(* CODESYS project Dashboard.project

Project tree, tasks and I/O mapping:
  Device : CODESYS Control for Raspberry Pi MC SL, CODESYS, order no. 2302000009, version 4.21.0.0
    application Application
      libraries: Standard, 3.5.22.0 (System); ifmEIP, 4.5.1.12 (ifm efector inc.); CAA Memory, * (CAA Technical Workgroup); CAA Can Low Level Extern, * (CAA Technical Workgroup); CmpBitmapPool, * (System)
      task VISU_TASK (cyclic, interval 100 ms, priority 31) calls VisuElems.Visu_Prg
      task MainTask (cyclic, interval t#20ms, priority 1) calls Main
      task ENIPScannerIOTask (cyclic, interval t#10ms, priority 0) calls EtherNet_IP_Scanner.IOCycle
      task ENIPScannerServiceTask (cyclic, interval t#20ms, priority 30) calls EtherNet_IP_Scanner.ServiceCycle
      program Main [ST]
      image pool Logo
      visualisation Connected_Devices_Dashboard
      global variables GL_Variables
      function block IOLink_Dashboard [FBD]: Process_Data, Dashboard_Data
    Onewire
    Ethernet : Ethernet, CODESYS, version 4.2.0.0
        settings: IPAddress = [192,168,1,99]; SubnetMask = [255,255,255,0]; GatewayAddress = [192,168,1,102]; MACAddress = [16#B8,16#27,16#EB,16#2F,16#E3,16#0E]; NetworkInterfaceName = 'eth0'; NetworkInterfaceName = "eth0"; SaveCommunicationSettings = FALSE; IPAddress = [192,168,0,2]; SubnetMask = [255,255,255,0]; GatewayAddress = [0,0,0,0]
      EtherNet_IP_Scanner : EtherNet/IP Scanner, CODESYS, order no. 1, version 4.9.0.0
        AL1423 : IO-Link Master PFL EIP 8P IP69K, ifm electronic, order no. AL1423, version Major Revision=16#2, Minor Revision = 16#3
            settings: INITIALIZED = TRUE; IP address of Target = [16#C0,16#A8,16#01,16#C8]; Keying.Check Minor Revision = FALSE; RequiredConfigVersion = 50660864; Number of Connections = 1; Connection Settings.Requested packet intervall = 10000 µs; Connection Settings.OT Connection Parameters = 18740; Connection Settings.TO Connection Parameters = 18880; Connection Settings.Connection Flags = 1056; Connection Settings.Connection Path Size = 8; Connection Settings.Config#2 Size = 130; Connection Settings.Large OT Connection Parameters = 1207959860; Connection Settings.Large TO Connection Parameters = 1207960000; Heartbeat Multiplier = 1; Input Data.ReadOnly = False; Input Data.BitSize = 16; Input Data.DataSize = 2; Input Data.ReadOnly = False; Input Data.BitSize = 16; Input Data.DataSize = 2; Input Data.ReadOnly = False; Input Data.BitSize = 16; Input Data.DataSize = 2; Input Data.ReadOnly = False; Input Data.BitSize = 16; Input Data.DataSize = 2; Input Data.ReadOnly = False; Input Data.BitSize = 16; Input Data.DataSize = 2; Input Data.ReadOnly = False; Input Data.BitSize = 16; Input Data.DataSize = 2; Input Data.ReadOnly = False; Input Data.BitSize = 16; Input Data.DataSize = 2; Input Data.ReadOnly = False; Input Data.BitSize = 16; Input Data.DataSize = 2; Input Data.ReadOnly = False; Input Data.BitSize = 16;
              Input Data.DataSize = 2; Input Data.ReadOnly = False; Input Data.BitSize = 16; Input Data.DataSize = 2; Input Data.ReadOnly = False; Input Data.BitSize = 16; Input Data.DataSize = 2; Input Data.ReadOnly = False; Input Data.BitSize = 16; Input Data.DataSize = 2; Input Data.ReadOnly = False; Input Data.BitSize = 16; Input Data.DataSize = 2; Input Data.ReadOnly = False; Input Data.BitSize = 16; Input Data.DataSize = 2; Input Data.ReadOnly = False; Input Data.BitSize = 16; Input Data.DataSize = 2; Input Data.ReadOnly = False; Input Data.BitSize = 16; Input Data.DataSize = 2; Input Data.ReadOnly = False; Input Data.BitSize = 16; Input Data.DataSize = 2; Input Data.ReadOnly = False; Input Data.BitSize = 16; Input Data.DataSize = 2; Input Data.ReadOnly = False; Input Data.BitSize = 16; Input Data.DataSize = 2; Input Data.ReadOnly = False; Input Data.BitSize = 16; Input Data.DataSize = 2; Input Data.ReadOnly = False; Input Data.BitSize = 16; Input Data.DataSize = 2; Input Data.ReadOnly = False; Input Data.BitSize = 16; Input Data.DataSize = 2;
              Input Data.ReadOnly = False; Input Data.BitSize = 16; Input Data.DataSize = 2; Input Data.ReadOnly = False; Input Data.BitSize = 16; Input Data.DataSize = 2; Input Data.ReadOnly = False; Input Data.BitSize = 16; Input Data.DataSize = 2; Input Data.ReadOnly = False; Input Data.BitSize = 16; Input Data.DataSize = 2; Input Data.ReadOnly = False; Input Data.BitSize = 16; Input Data.DataSize = 2; Input Data.ReadOnly = False; Input Data.BitSize = 16; Input Data.DataSize = 2; Input Data.ReadOnly = False; Input Data.BitSize = 16; Input Data.DataSize = 2; Input Data.ReadOnly = False; Input Data.BitSize = 16; Input Data.DataSize = 2; Input Data.ReadOnly = False; Input Data.BitSize = 16; Input Data.DataSize = 2; Input Data.ReadOnly = False; Input Data.BitSize = 16; Input Data.DataSize = 2; Input Data.ReadOnly = False; Input Data.BitSize = 16; Input Data.DataSize = 2; Input Data.ReadOnly = False; Input Data.BitSize = 16; Input Data.DataSize = 2; Input Data.ReadOnly = False; Input Data.BitSize = 16; Input Data.DataSize = 2; Input Data.ReadOnly = False;
              Input Data.BitSize = 16; Input Data.DataSize = 2; Input Data.ReadOnly = False; Input Data.BitSize = 16; Input Data.DataSize = 2; Input Data.ReadOnly = False; Input Data.BitSize = 16; Input Data.DataSize = 2; Input Data.ReadOnly = False; Input Data.BitSize = 16; Input Data.DataSize = 2; Input Data.ReadOnly = False; Input Data.BitSize = 16; Input Data.DataSize = 2; Input Data.ReadOnly = False; Input Data.BitSize = 16; Input Data.DataSize = 2; Input Data.ReadOnly = False; Input Data.BitSize = 16; Input Data.DataSize = 2; Input Data.ReadOnly = False; Input Data.BitSize = 16; Input Data.DataSize = 2; Input Data.ReadOnly = False; Input Data.BitSize = 16; Input Data.DataSize = 2; Input Data.ReadOnly = False; Input Data.BitSize = 16; Input Data.DataSize = 2; Input Data.ReadOnly = False; Input Data.BitSize = 16; Input Data.DataSize = 2; Input Data.ReadOnly = False; Input Data.BitSize = 16; Input Data.DataSize = 2; Input Data.ReadOnly = False; Input Data.BitSize = 16; Input Data.DataSize = 2; Input Data.ReadOnly = False; Input Data.BitSize = 16;
              Input Data.DataSize = 2; Input Data.ReadOnly = False; Input Data.BitSize = 16; Input Data.DataSize = 2; Input Data.ReadOnly = False; Input Data.BitSize = 16; Input Data.DataSize = 2; Input Data.ReadOnly = False; Input Data.BitSize = 16; Input Data.DataSize = 2; Input Data.ReadOnly = False; Input Data.BitSize = 16; Input Data.DataSize = 2; Input Data.ReadOnly = False; Input Data.BitSize = 16; Input Data.DataSize = 2; Input Data.ReadOnly = False; Input Data.BitSize = 16; Input Data.DataSize = 2; Input Data.ReadOnly = False; Input Data.BitSize = 16; Input Data.DataSize = 2; Input Data.ReadOnly = False; Input Data.BitSize = 16; Input Data.DataSize = 2; Input Data.ReadOnly = False; Input Data.BitSize = 16; Input Data.DataSize = 2; Input Data.ReadOnly = False; Input Data.BitSize = 16; Input Data.DataSize = 2; Input Data.ReadOnly = False; Input Data.BitSize = 16; Input Data.DataSize = 2; Input Data.ReadOnly = False; Input Data.BitSize = 16; Input Data.DataSize = 2; Input Data.ReadOnly = False; Input Data.BitSize = 16; Input Data.DataSize = 2;
              Input Data.ReadOnly = False; Input Data.BitSize = 16; Input Data.DataSize = 2; Input Data.ReadOnly = False; Input Data.BitSize = 16; Input Data.DataSize = 2; Input Data.ReadOnly = False; Input Data.BitSize = 16; Input Data.DataSize = 2; Input Data.ReadOnly = False; Input Data.BitSize = 16; Input Data.DataSize = 2; Input Data.ReadOnly = False; Input Data.BitSize = 16; Input Data.DataSize = 2; Input Data.ReadOnly = False; Input Data.BitSize = 16; Input Data.DataSize = 2; Input Data.ReadOnly = False; Input Data.BitSize = 16; Input Data.DataSize = 2; Input Data.ReadOnly = False; Input Data.BitSize = 16; Input Data.DataSize = 2; Input Data.ReadOnly = False; Input Data.BitSize = 16; Input Data.DataSize = 2; Input Data.ReadOnly = False; Input Data.BitSize = 16; Input Data.DataSize = 2; Input Data.ReadOnly = False; Input Data.BitSize = 16; Input Data.DataSize = 2; Input Data.ReadOnly = False; Input Data.BitSize = 16; Input Data.DataSize = 2; Input Data.ReadOnly = False; Input Data.BitSize = 16; Input Data.DataSize = 2; Input Data.ReadOnly = False;
              Input Data.BitSize = 16; Input Data.DataSize = 2; Input Data.ReadOnly = False; Input Data.BitSize = 16; Input Data.DataSize = 2; Input Data.ReadOnly = False; Input Data.BitSize = 16; Input Data.DataSize = 2; Input Data.ReadOnly = False; Input Data.BitSize = 16; Input Data.DataSize = 2; Input Data.ReadOnly = False; Input Data.BitSize = 16; Input Data.DataSize = 2; Input Data.ReadOnly = False; Input Data.BitSize = 16; Input Data.DataSize = 2; Input Data.ReadOnly = False; Input Data.BitSize = 16; Input Data.DataSize = 2; Input Data.ReadOnly = False; Input Data.BitSize = 16; Input Data.DataSize = 2; Input Data.ReadOnly = False; Input Data.BitSize = 16; Input Data.DataSize = 2; Input Data.ReadOnly = False; Input Data.BitSize = 16; Input Data.DataSize = 2; Input Data.ReadOnly = False; Input Data.BitSize = 16; Input Data.DataSize = 2; Input Data.ReadOnly = False; Input Data.BitSize = 16; Input Data.DataSize = 2; Input Data.ReadOnly = False; Input Data.BitSize = 16; Input Data.DataSize = 2; Input Data.ReadOnly = False; Input Data.BitSize = 16;
              Input Data.DataSize = 2; Input Data.ReadOnly = False; Input Data.BitSize = 16; Input Data.DataSize = 2; Input Data.ReadOnly = False; Input Data.BitSize = 16; Input Data.DataSize = 2; Input Data.ReadOnly = False; Input Data.BitSize = 16; Input Data.DataSize = 2; Input Data.ReadOnly = False; Input Data.BitSize = 16; Input Data.DataSize = 2; Input Data.ReadOnly = False; Input Data.BitSize = 16; Input Data.DataSize = 2; Input Data.ReadOnly = False; Input Data.BitSize = 16; Input Data.DataSize = 2; Input Data.ReadOnly = False; Input Data.BitSize = 16; Input Data.DataSize = 2; Input Data.ReadOnly = False; Input Data.BitSize = 16; Input Data.DataSize = 2; Input Data.ReadOnly = False; Input Data.BitSize = 16; Input Data.DataSize = 2; Input Data.ReadOnly = False; Input Data.BitSize = 16; Input Data.DataSize = 2; Input Data.ReadOnly = False; Input Data.BitSize = 16; Input Data.DataSize = 2; Input Data.ReadOnly = False; Input Data.BitSize = 16; Input Data.DataSize = 2; Input Data.ReadOnly = False; Input Data.BitSize = 16; Input Data.DataSize = 2;
              Input Data.ReadOnly = False; Input Data.BitSize = 16; Input Data.DataSize = 2; Input Data.ReadOnly = False; Input Data.BitSize = 16; Input Data.DataSize = 2; Input Data.ReadOnly = False; Input Data.BitSize = 16; Input Data.DataSize = 2; Input Data.ReadOnly = False; Input Data.BitSize = 16; Input Data.DataSize = 2; Input Data.ReadOnly = False; Input Data.BitSize = 16; Input Data.DataSize = 2; Input Data.ReadOnly = False; Input Data.BitSize = 16; Input Data.DataSize = 2; Input Data.ReadOnly = False; Input Data.BitSize = 16; Input Data.DataSize = 2; Input Data.ReadOnly = False; Input Data.BitSize = 16; Input Data.DataSize = 2; Input Data.ReadOnly = False; Input Data.BitSize = 16; Input Data.DataSize = 2; Input Data.ReadOnly = False; Input Data.BitSize = 16; Input Data.DataSize = 2; Input Data.ReadOnly = False; Input Data.BitSize = 16; Input Data.DataSize = 2; Input Data.ReadOnly = False; Input Data.BitSize = 16; Input Data.DataSize = 2; Input Data.ReadOnly = False; Input Data.BitSize = 16; Input Data.DataSize = 2; Input Data.ReadOnly = False;
              Input Data.BitSize = 16; Input Data.DataSize = 2; Input Data.ReadOnly = False; Input Data.BitSize = 16; Input Data.DataSize = 2; Input Data.ReadOnly = False; Input Data.BitSize = 16; Input Data.DataSize = 2; Input Data.ReadOnly = False; Input Data.BitSize = 16; Input Data.DataSize = 2; Input Data.ReadOnly = False; Input Data.BitSize = 16; Input Data.DataSize = 2; Input Data.ReadOnly = False; Input Data.BitSize = 16; Input Data.DataSize = 2; Input Data.ReadOnly = False; Input Data.BitSize = 16; Input Data.DataSize = 2; Input Data.ReadOnly = False; Input Data.BitSize = 16; Input Data.DataSize = 2; Input Data.ReadOnly = False; Input Data.BitSize = 16; Input Data.DataSize = 2; Input Data.ReadOnly = False; Input Data.BitSize = 16; Input Data.DataSize = 2; Input Data.ReadOnly = False; Input Data.BitSize = 16; Input Data.DataSize = 2; Input Data.ReadOnly = False; Input Data.BitSize = 16; Input Data.DataSize = 2; Input Data.ReadOnly = False; Input Data.BitSize = 16; Input Data.DataSize = 2; Input Data.ReadOnly = False; Input Data.BitSize = 16;
              Input Data.DataSize = 2; Input Data.ReadOnly = False; Input Data.BitSize = 16; Input Data.DataSize = 2; Input Data.ReadOnly = False; Input Data.BitSize = 16; Input Data.DataSize = 2; Input Data.ReadOnly = False; Input Data.BitSize = 16; Input Data.DataSize = 2; Input Data.ReadOnly = False; Input Data.BitSize = 16; Input Data.DataSize = 2; Input Data.ReadOnly = False; Input Data.BitSize = 16; Input Data.DataSize = 2; Input Data.ReadOnly = False; Input Data.BitSize = 16; Input Data.DataSize = 2; Input Data.ReadOnly = False; Input Data.BitSize = 16; Input Data.DataSize = 2; Input Data.ReadOnly = False; Input Data.BitSize = 16; Input Data.DataSize = 2; Input Data.ReadOnly = False; Input Data.BitSize = 16; Input Data.DataSize = 2; Input Data.ReadOnly = False; Input Data.BitSize = 16; Input Data.DataSize = 2; Input Data.ReadOnly = False; Input Data.BitSize = 16; Input Data.DataSize = 2; Input Data.ReadOnly = False; Input Data.BitSize = 16; Input Data.DataSize = 2; Input Data.ReadOnly = False; Input Data.BitSize = 16; Input Data.DataSize = 2;
              Input Data.ReadOnly = False; Input Data.BitSize = 16; Input Data.DataSize = 2; Input Data.ReadOnly = False; Input Data.BitSize = 16; Input Data.DataSize = 2; Input Data.ReadOnly = False; Input Data.BitSize = 16; Input Data.DataSize = 2; Input Data.ReadOnly = False; Input Data.BitSize = 16; Input Data.DataSize = 2; Input Data.ReadOnly = False; Input Data.BitSize = 16; Input Data.DataSize = 2; Input Data.ReadOnly = False; Input Data.BitSize = 16; Input Data.DataSize = 2; Input Data.ReadOnly = False; Input Data.BitSize = 16; Input Data.DataSize = 2; Input Data.ReadOnly = False; Input Data.BitSize = 16; Input Data.DataSize = 2; Input Data.ReadOnly = False; Input Data.BitSize = 16; Input Data.DataSize = 2; Input Data.ReadOnly = False; Input Data.BitSize = 16; Input Data.DataSize = 2; Input Data.ReadOnly = False; Input Data.BitSize = 16; Input Data.DataSize = 2; Input Data.ReadOnly = False; Input Data.BitSize = 16; Input Data.DataSize = 2; Input Data.ReadOnly = False; Input Data.BitSize = 16; Input Data.DataSize = 2; Input Data.ReadOnly = False;
              Input Data.BitSize = 16; Input Data.DataSize = 2; Input Data.ReadOnly = False; Input Data.BitSize = 16; Input Data.DataSize = 2; Input Data.ReadOnly = False; Input Data.BitSize = 16; Input Data.DataSize = 2; Input Data.ReadOnly = False; Input Data.BitSize = 16; Input Data.DataSize = 2; Input Data.ReadOnly = False; Input Data.BitSize = 16; Input Data.DataSize = 2; Input Data.ReadOnly = False; Input Data.BitSize = 16; Input Data.DataSize = 2; Input Data.ReadOnly = False; Input Data.BitSize = 16; Input Data.DataSize = 2; Input Data.ReadOnly = False; Input Data.BitSize = 16; Input Data.DataSize = 2; Input Data.ReadOnly = False; Input Data.BitSize = 16; Input Data.DataSize = 2; Input Data.ReadOnly = False; Input Data.BitSize = 16; Input Data.DataSize = 2; Input Data.ReadOnly = False; Input Data.BitSize = 16; Input Data.DataSize = 2; Input Data.ReadOnly = False; Input Data.BitSize = 16; Input Data.DataSize = 2; Input Data.ReadOnly = False; Input Data.BitSize = 16; Input Data.DataSize = 2; Input Data.ReadOnly = False; Input Data.BitSize = 16;
              Input Data.DataSize = 2; Input Data.ReadOnly = False; Input Data.BitSize = 16; Input Data.DataSize = 2; Input Data.ReadOnly = False; Input Data.BitSize = 16; Input Data.DataSize = 2; Input Data.ReadOnly = False; Input Data.BitSize = 16; Input Data.DataSize = 2; Input Data.ReadOnly = False; Input Data.BitSize = 16; Input Data.DataSize = 2; Input Data.ReadOnly = False; Input Data.BitSize = 16; Input Data.DataSize = 2; Input Data.ReadOnly = False; Input Data.BitSize = 16; Input Data.DataSize = 2; Input Data.ReadOnly = False; Input Data.BitSize = 16; Input Data.DataSize = 2; Input Data.ReadOnly = False; Input Data.BitSize = 16; Input Data.DataSize = 2; Input Data.ReadOnly = False; Input Data.BitSize = 16; Input Data.DataSize = 2; Input Data.ReadOnly = False; Input Data.BitSize = 16; Input Data.DataSize = 2; Input Data.ReadOnly = False; Input Data.BitSize = 16; Input Data.DataSize = 2; Input Data.ReadOnly = False; Input Data.BitSize = 16; Input Data.DataSize = 2; Input Data.ReadOnly = False; Input Data.BitSize = 16; Input Data.DataSize = 2;
              Input Data.ReadOnly = False; Input Data.BitSize = 16; Input Data.DataSize = 2; Input Data.ReadOnly = False; Input Data.BitSize = 16; Input Data.DataSize = 2; Input Data.ReadOnly = False; Input Data.BitSize = 16; Input Data.DataSize = 2; Input Data.ReadOnly = False; Input Data.BitSize = 16; Input Data.DataSize = 2; Input Data.ReadOnly = False; Input Data.BitSize = 16; Input Data.DataSize = 2; Input Data.ReadOnly = False; Input Data.BitSize = 16; Input Data.DataSize = 2; Input Data.ReadOnly = False; Input Data.BitSize = 16; Input Data.DataSize = 2; Input Data.ReadOnly = False; Input Data.BitSize = 16; Input Data.DataSize = 2; Input Data.ReadOnly = False; Input Data.BitSize = 16; Input Data.DataSize = 2; Input Data.ReadOnly = False; Input Data.BitSize = 16; Input Data.DataSize = 2; Input Data.ReadOnly = False; Input Data.BitSize = 16; Input Data.DataSize = 2; Input Data.ReadOnly = False; Input Data.BitSize = 16; Input Data.DataSize = 2; Input Data.ReadOnly = False; Input Data.BitSize = 16; Input Data.DataSize = 2; Input Data.ReadOnly = False;
              Input Data.BitSize = 16; Input Data.DataSize = 2; Input Data.ReadOnly = False; Input Data.BitSize = 16; Input Data.DataSize = 2; Input Data.ReadOnly = False; Input Data.BitSize = 16; Input Data.DataSize = 2; Input Data.ReadOnly = False; Input Data.BitSize = 16; Input Data.DataSize = 2; Input Data.ReadOnly = False; Input Data.BitSize = 16; Input Data.DataSize = 2; Input Data.ReadOnly = False; Input Data.BitSize = 16; Input Data.DataSize = 2; Input Data.ReadOnly = False; Input Data.BitSize = 16; Input Data.DataSize = 2; Input Data.ReadOnly = False; Input Data.BitSize = 16; Input Data.DataSize = 2; Input Data.ReadOnly = False; Input Data.BitSize = 16; Input Data.DataSize = 2; Input Data.ReadOnly = False; Input Data.BitSize = 16; Input Data.DataSize = 2; Input Data.ReadOnly = False; Input Data.BitSize = 16; Input Data.DataSize = 2; Input Data.ReadOnly = False; Input Data.BitSize = 16; Input Data.DataSize = 2; Input Data.ReadOnly = False; Input Data.BitSize = 16; Input Data.DataSize = 2; Input Data.ReadOnly = False; Input Data.BitSize = 16;
              Input Data.DataSize = 2; Input Data.ReadOnly = False; Input Data.BitSize = 16; Input Data.DataSize = 2; Input Data.ReadOnly = False; Input Data.BitSize = 16; Input Data.DataSize = 2; Input Data.ReadOnly = False; Input Data.BitSize = 16; Input Data.DataSize = 2; Input Data.ReadOnly = False; Input Data.BitSize = 16; Input Data.DataSize = 2; Input Data.ReadOnly = False; Input Data.BitSize = 16; Input Data.DataSize = 2; Input Data.ReadOnly = False; Input Data.BitSize = 16; Input Data.DataSize = 2; Input Data.ReadOnly = False; Input Data.BitSize = 16; Input Data.DataSize = 2; Input Data.ReadOnly = False; Input Data.BitSize = 16; Input Data.DataSize = 2; Input Data.ReadOnly = False; Input Data.BitSize = 16; Input Data.DataSize = 2; Input Data.ReadOnly = False; Input Data.BitSize = 16; Input Data.DataSize = 2; Input Data.ReadOnly = False; Input Data.BitSize = 16; Input Data.DataSize = 2; Input Data.ReadOnly = False; Input Data.BitSize = 16; Input Data.DataSize = 2; Input Data.ReadOnly = False; Input Data.BitSize = 16; Input Data.DataSize = 2;
              Input Data.ReadOnly = False; Input Data.BitSize = 16; Input Data.DataSize = 2; Output Data.ReadOnly = False; Output Data.BitSize = 16; Output Data.DataSize = 2; Output Data.ReadOnly = False; Output Data.BitSize = 16; Output Data.DataSize = 2; Output Data.ReadOnly = False; Output Data.BitSize = 16; Output Data.DataSize = 2; Output Data.ReadOnly = False; Output Data.BitSize = 16; Output Data.DataSize = 2; Output Data.ReadOnly = False; Output Data.BitSize = 16; Output Data.DataSize = 2; Output Data.ReadOnly = False; Output Data.BitSize = 16; Output Data.DataSize = 2; Output Data.ReadOnly = False; Output Data.BitSize = 16; Output Data.DataSize = 2; Output Data.ReadOnly = False; Output Data.BitSize = 16; Output Data.DataSize = 2; Output Data.ReadOnly = False; Output Data.BitSize = 16; Output Data.DataSize = 2; Output Data.ReadOnly = False; Output Data.BitSize = 16; Output Data.DataSize = 2; Output Data.ReadOnly = False; Output Data.BitSize = 16; Output Data.DataSize = 2; Output Data.ReadOnly = False; Output Data.BitSize = 16; Output Data.DataSize = 2; Output Data.ReadOnly = False;
              Output Data.BitSize = 16; Output Data.DataSize = 2; Output Data.ReadOnly = False; Output Data.BitSize = 16; Output Data.DataSize = 2; Output Data.ReadOnly = False; Output Data.BitSize = 16; Output Data.DataSize = 2; Output Data.ReadOnly = False; Output Data.BitSize = 16; Output Data.DataSize = 2; Output Data.ReadOnly = False; Output Data.BitSize = 16; Output Data.DataSize = 2; Output Data.ReadOnly = False; Output Data.BitSize = 16; Output Data.DataSize = 2; Output Data.ReadOnly = False; Output Data.BitSize = 16; Output Data.DataSize = 2; Output Data.ReadOnly = False; Output Data.BitSize = 16; Output Data.DataSize = 2; Output Data.ReadOnly = False; Output Data.BitSize = 16; Output Data.DataSize = 2; Output Data.ReadOnly = False; Output Data.BitSize = 16; Output Data.DataSize = 2; Output Data.ReadOnly = False; Output Data.BitSize = 16; Output Data.DataSize = 2; Output Data.ReadOnly = False; Output Data.BitSize = 16; Output Data.DataSize = 2; Output Data.ReadOnly = False; Output Data.BitSize = 16; Output Data.DataSize = 2; Output Data.ReadOnly = False; Output Data.BitSize = 16;
              Output Data.DataSize = 2; Output Data.ReadOnly = False; Output Data.BitSize = 16; Output Data.DataSize = 2; Output Data.ReadOnly = False; Output Data.BitSize = 16; Output Data.DataSize = 2; Output Data.ReadOnly = False; Output Data.BitSize = 16; Output Data.DataSize = 2; Output Data.ReadOnly = False; Output Data.BitSize = 16; Output Data.DataSize = 2; Output Data.ReadOnly = False; Output Data.BitSize = 16; Output Data.DataSize = 2; Output Data.ReadOnly = False; Output Data.BitSize = 16; Output Data.DataSize = 2; Output Data.ReadOnly = False; Output Data.BitSize = 16; Output Data.DataSize = 2; Output Data.ReadOnly = False; Output Data.BitSize = 16; Output Data.DataSize = 2; Output Data.ReadOnly = False; Output Data.BitSize = 16; Output Data.DataSize = 2; Output Data.ReadOnly = False; Output Data.BitSize = 16; Output Data.DataSize = 2; Output Data.ReadOnly = False; Output Data.BitSize = 16; Output Data.DataSize = 2; Output Data.ReadOnly = False; Output Data.BitSize = 16; Output Data.DataSize = 2; Output Data.ReadOnly = False; Output Data.BitSize = 16; Output Data.DataSize = 2;
              Output Data.ReadOnly = False; Output Data.BitSize = 16; Output Data.DataSize = 2; Output Data.ReadOnly = False; Output Data.BitSize = 16; Output Data.DataSize = 2; Output Data.ReadOnly = False; Output Data.BitSize = 16; Output Data.DataSize = 2; Output Data.ReadOnly = False; Output Data.BitSize = 16; Output Data.DataSize = 2; Output Data.ReadOnly = False; Output Data.BitSize = 16; Output Data.DataSize = 2; Output Data.ReadOnly = False; Output Data.BitSize = 16; Output Data.DataSize = 2; Output Data.ReadOnly = False; Output Data.BitSize = 16; Output Data.DataSize = 2; Output Data.ReadOnly = False; Output Data.BitSize = 16; Output Data.DataSize = 2; Output Data.ReadOnly = False; Output Data.BitSize = 16; Output Data.DataSize = 2; Output Data.ReadOnly = False; Output Data.BitSize = 16; Output Data.DataSize = 2; Output Data.ReadOnly = False; Output Data.BitSize = 16; Output Data.DataSize = 2; Output Data.ReadOnly = False; Output Data.BitSize = 16; Output Data.DataSize = 2; Output Data.ReadOnly = False; Output Data.BitSize = 16; Output Data.DataSize = 2; Output Data.ReadOnly = False;
              Output Data.BitSize = 16; Output Data.DataSize = 2; Output Data.ReadOnly = False; Output Data.BitSize = 16; Output Data.DataSize = 2; Output Data.ReadOnly = False; Output Data.BitSize = 16; Output Data.DataSize = 2; Output Data.ReadOnly = False; Output Data.BitSize = 16; Output Data.DataSize = 2; Output Data.ReadOnly = False; Output Data.BitSize = 16; Output Data.DataSize = 2; Output Data.ReadOnly = False; Output Data.BitSize = 16; Output Data.DataSize = 2; Output Data.ReadOnly = False; Output Data.BitSize = 16; Output Data.DataSize = 2; Output Data.ReadOnly = False; Output Data.BitSize = 16; Output Data.DataSize = 2; Output Data.ReadOnly = False; Output Data.BitSize = 16; Output Data.DataSize = 2; Output Data.ReadOnly = False; Output Data.BitSize = 16; Output Data.DataSize = 2; Output Data.ReadOnly = False; Output Data.BitSize = 16; Output Data.DataSize = 2; Output Data.ReadOnly = False; Output Data.BitSize = 16; Output Data.DataSize = 2; Output Data.ReadOnly = False; Output Data.BitSize = 16; Output Data.DataSize = 2; Output Data.ReadOnly = False; Output Data.BitSize = 16;
              Output Data.DataSize = 2; Output Data.ReadOnly = False; Output Data.BitSize = 16; Output Data.DataSize = 2; Output Data.ReadOnly = False; Output Data.BitSize = 16; Output Data.DataSize = 2; Output Data.ReadOnly = False; Output Data.BitSize = 16; Output Data.DataSize = 2; Output Data.ReadOnly = False; Output Data.BitSize = 16; Output Data.DataSize = 2; Output Data.ReadOnly = False; Output Data.BitSize = 16; Output Data.DataSize = 2; Output Data.ReadOnly = False; Output Data.BitSize = 16; Output Data.DataSize = 2; Output Data.ReadOnly = False; Output Data.BitSize = 16; Output Data.DataSize = 2; Output Data.ReadOnly = False; Output Data.BitSize = 16; Output Data.DataSize = 2; Output Data.ReadOnly = False; Output Data.BitSize = 16; Output Data.DataSize = 2; Output Data.ReadOnly = False; Output Data.BitSize = 16; Output Data.DataSize = 2; Output Data.ReadOnly = False; Output Data.BitSize = 16; Output Data.DataSize = 2; Output Data.ReadOnly = False; Output Data.BitSize = 16; Output Data.DataSize = 2; Output Data.ReadOnly = False; Output Data.BitSize = 16; Output Data.DataSize = 2;
              Output Data.ReadOnly = False; Output Data.BitSize = 16; Output Data.DataSize = 2; Output Data.ReadOnly = False; Output Data.BitSize = 16; Output Data.DataSize = 2; Output Data.ReadOnly = False; Output Data.BitSize = 16; Output Data.DataSize = 2; Output Data.ReadOnly = False; Output Data.BitSize = 16; Output Data.DataSize = 2; Output Data.ReadOnly = False; Output Data.BitSize = 16; Output Data.DataSize = 2; Output Data.ReadOnly = False; Output Data.BitSize = 16; Output Data.DataSize = 2; Output Data.ReadOnly = False; Output Data.BitSize = 16; Output Data.DataSize = 2; Output Data.ReadOnly = False; Output Data.BitSize = 16; Output Data.DataSize = 2; Output Data.ReadOnly = False; Output Data.BitSize = 16; Output Data.DataSize = 2; Output Data.ReadOnly = False; Output Data.BitSize = 16; Output Data.DataSize = 2; Output Data.ReadOnly = False; Output Data.BitSize = 16; Output Data.DataSize = 2; Output Data.ReadOnly = False; Output Data.BitSize = 16; Output Data.DataSize = 2; Output Data.ReadOnly = False; Output Data.BitSize = 16; Output Data.DataSize = 2; Output Data.ReadOnly = False;
              Output Data.BitSize = 16; Output Data.DataSize = 2; Output Data.ReadOnly = False; Output Data.BitSize = 16; Output Data.DataSize = 2; Output Data.ReadOnly = False; Output Data.BitSize = 16; Output Data.DataSize = 2; Output Data.ReadOnly = False; Output Data.BitSize = 16; Output Data.DataSize = 2; Output Data.ReadOnly = False; Output Data.BitSize = 16; Output Data.DataSize = 2; Output Data.ReadOnly = False; Output Data.BitSize = 16; Output Data.DataSize = 2; Output Data.ReadOnly = False; Output Data.BitSize = 16; Output Data.DataSize = 2; Output Data.ReadOnly = False; Output Data.BitSize = 16; Output Data.DataSize = 2; Output Data.ReadOnly = False; Output Data.BitSize = 16; Output Data.DataSize = 2; Output Data.ReadOnly = False; Output Data.BitSize = 16; Output Data.DataSize = 2; Output Data.ReadOnly = False; Output Data.BitSize = 16; Output Data.DataSize = 2; Output Data.ReadOnly = False; Output Data.BitSize = 16; Output Data.DataSize = 2; Output Data.ReadOnly = False; Output Data.BitSize = 16; Output Data.DataSize = 2; Output Data.ReadOnly = False; Output Data.BitSize = 16;
              Output Data.DataSize = 2; Output Data.ReadOnly = False; Output Data.BitSize = 16; Output Data.DataSize = 2; Output Data.ReadOnly = False; Output Data.BitSize = 16; Output Data.DataSize = 2; Output Data.ReadOnly = False; Output Data.BitSize = 16; Output Data.DataSize = 2; Output Data.ReadOnly = False; Output Data.BitSize = 16; Output Data.DataSize = 2; Output Data.ReadOnly = False; Output Data.BitSize = 16; Output Data.DataSize = 2; Output Data.ReadOnly = False; Output Data.BitSize = 16; Output Data.DataSize = 2; Output Data.ReadOnly = False; Output Data.BitSize = 16; Output Data.DataSize = 2; Output Data.ReadOnly = False; Output Data.BitSize = 16; Output Data.DataSize = 2; Output Data.ReadOnly = False; Output Data.BitSize = 16; Output Data.DataSize = 2; Output Data.ReadOnly = False; Output Data.BitSize = 16; Output Data.DataSize = 2; Output Data.ReadOnly = False; Output Data.BitSize = 16; Output Data.DataSize = 2; Output Data.ReadOnly = False; Output Data.BitSize = 16; Output Data.DataSize = 2; Output Data.ReadOnly = False; Output Data.BitSize = 16; Output Data.DataSize = 2;
              Output Data.ReadOnly = False; Output Data.BitSize = 16; Output Data.DataSize = 2; Output Data.ReadOnly = False; Output Data.BitSize = 16; Output Data.DataSize = 2; Output Data.ReadOnly = False; Output Data.BitSize = 16; Output Data.DataSize = 2; Output Data.ReadOnly = False; Output Data.BitSize = 16; Output Data.DataSize = 2; Output Data.ReadOnly = False; Output Data.BitSize = 16; Output Data.DataSize = 2; Output Data.ReadOnly = False; Output Data.BitSize = 16; Output Data.DataSize = 2; Output Data.ReadOnly = False; Output Data.BitSize = 16; Output Data.DataSize = 2; Output Data.ReadOnly = False; Output Data.BitSize = 16; Output Data.DataSize = 2; Output Data.ReadOnly = False; Output Data.BitSize = 16; Output Data.DataSize = 2; Output Data.ReadOnly = False; Output Data.BitSize = 16; Output Data.DataSize = 2; Output Data.ReadOnly = False; Output Data.BitSize = 16; Output Data.DataSize = 2; Output Data.ReadOnly = False; Output Data.BitSize = 16; Output Data.DataSize = 2; Output Data.ReadOnly = False; Output Data.BitSize = 16; Output Data.DataSize = 2; Output Data.ReadOnly = False;
              Output Data.BitSize = 16; Output Data.DataSize = 2; Output Data.ReadOnly = False; Output Data.BitSize = 16; Output Data.DataSize = 2; Output Data.ReadOnly = False; Output Data.BitSize = 16; Output Data.DataSize = 2; Output Data.ReadOnly = False; Output Data.BitSize = 16; Output Data.DataSize = 2; Output Data.ReadOnly = False; Output Data.BitSize = 16; Output Data.DataSize = 2; Output Data.ReadOnly = False; Output Data.BitSize = 16; Output Data.DataSize = 2; Output Data.ReadOnly = False; Output Data.BitSize = 16; Output Data.DataSize = 2; Output Data.ReadOnly = False; Output Data.BitSize = 16; Output Data.DataSize = 2; Output Data.ReadOnly = False; Output Data.BitSize = 16; Output Data.DataSize = 2; Output Data.ReadOnly = False; Output Data.BitSize = 16; Output Data.DataSize = 2; Output Data.ReadOnly = False; Output Data.BitSize = 16; Output Data.DataSize = 2; Output Data.ReadOnly = False; Output Data.BitSize = 16; Output Data.DataSize = 2; Output Data.ReadOnly = False; Output Data.BitSize = 16; Output Data.DataSize = 2; Output Data.ReadOnly = False; Output Data.BitSize = 16;
              Output Data.DataSize = 2; Output Data.ReadOnly = False; Output Data.BitSize = 16; Output Data.DataSize = 2; Output Data.ReadOnly = False; Output Data.BitSize = 16; Output Data.DataSize = 2; Output Data.ReadOnly = False; Output Data.BitSize = 16; Output Data.DataSize = 2; Output Data.ReadOnly = False; Output Data.BitSize = 16; Output Data.DataSize = 2; Output Data.ReadOnly = False; Output Data.BitSize = 16; Output Data.DataSize = 2; Input Data.Name = 'Input Data'; Input Data.HelpString = ''; Input Data.ReadOnly = False; Input Data.BitSize = 16; Input Data.DataSize = 2; Input Data.DataType = 'UINT'; Input Data.Name = 'Input Data'; Input Data.HelpString = ''; Input Data.ReadOnly = False; Input Data.BitSize = 16; Input Data.DataSize = 2; Input Data.DataType = 'UINT'; Input Data.Name = 'Input Data'; Input Data.HelpString = ''; Input Data.ReadOnly = False; Input Data.BitSize = 16; Input Data.DataSize = 2; Input Data.DataType = 'UINT'; Input Data.Name = 'Input Data'; Input Data.HelpString = ''; Input Data.ReadOnly = False; Input Data.BitSize = 16; Input Data.DataSize = 2; Input Data.DataType = 'UINT';
              Input Data.Name = 'Input Data'; Input Data.HelpString = ''; Input Data.ReadOnly = False; Input Data.BitSize = 16; Input Data.DataSize = 2; Input Data.DataType = 'UINT'; Input Data.Name = 'Input Data'; Input Data.HelpString = ''; Input Data.ReadOnly = False; Input Data.BitSize = 16; Input Data.DataSize = 2; Input Data.DataType = 'UINT'; Input Data.Name = 'Input Data'; Input Data.HelpString = ''; Input Data.ReadOnly = False; Input Data.BitSize = 16; Input Data.DataSize = 2; Input Data.DataType = 'UINT'; Input Data.Name = 'Input Data'; Input Data.HelpString = ''; Input Data.ReadOnly = False; Input Data.BitSize = 16; Input Data.DataSize = 2; Input Data.DataType = 'UINT'; Input Data.Name = 'Input Data'; Input Data.HelpString = ''; Input Data.ReadOnly = False; Input Data.BitSize = 16; Input Data.DataSize = 2; Input Data.DataType = 'UINT'; Input Data.Name = 'Input Data'; Input Data.HelpString = ''; Input Data.ReadOnly = False; Input Data.BitSize = 16; Input Data.DataSize = 2; Input Data.DataType = 'UINT'; Input Data.Name = 'Input Data'; Input Data.HelpString = ''; Input Data.ReadOnly = False; Input Data.BitSize = 16;
              Input Data.DataSize = 2; Input Data.DataType = 'UINT'; Input Data.Name = 'Input Data'; Input Data.HelpString = ''; Input Data.ReadOnly = False; Input Data.BitSize = 16; Input Data.DataSize = 2; Input Data.DataType = 'UINT'; Input Data.Name = 'Input Data'; Input Data.HelpString = ''; Input Data.ReadOnly = False; Input Data.BitSize = 16; Input Data.DataSize = 2; Input Data.DataType = 'UINT'; Input Data.Name = 'Input Data'; Input Data.HelpString = ''; Input Data.ReadOnly = False; Input Data.BitSize = 16; Input Data.DataSize = 2; Input Data.DataType = 'UINT'; Input Data.Name = 'Input Data'; Input Data.HelpString = ''; Input Data.ReadOnly = False; Input Data.BitSize = 16; Input Data.DataSize = 2; Input Data.DataType = 'UINT'; Input Data.Name = 'Input Data'; Input Data.HelpString = ''; Input Data.ReadOnly = False; Input Data.BitSize = 16; Input Data.DataSize = 2; Input Data.DataType = 'UINT'; Input Data.Name = 'Input Data'; Input Data.HelpString = ''; Input Data.ReadOnly = False; Input Data.BitSize = 16; Input Data.DataSize = 2; Input Data.DataType = 'UINT'; Input Data.Name = 'Input Data'; Input Data.HelpString = '';
              Input Data.ReadOnly = False; Input Data.BitSize = 16; Input Data.DataSize = 2; Input Data.DataType = 'UINT'; Input Data.Name = 'Input Data'; Input Data.HelpString = ''; Input Data.ReadOnly = False; Input Data.BitSize = 16; Input Data.DataSize = 2; Input Data.DataType = 'UINT'; Input Data.Name = 'Input Data'; Input Data.HelpString = ''; Input Data.ReadOnly = False; Input Data.BitSize = 16; Input Data.DataSize = 2; Input Data.DataType = 'UINT'; Input Data.Name = 'Input Data'; Input Data.HelpString = ''; Input Data.ReadOnly = False; Input Data.BitSize = 16; Input Data.DataSize = 2; Input Data.DataType = 'UINT'; Input Data.Name = 'Input Data'; Input Data.HelpString = ''; Input Data.ReadOnly = False; Input Data.BitSize = 16; Input Data.DataSize = 2; Input Data.DataType = 'UINT'; Input Data.Name = 'Input Data'; Input Data.HelpString = ''; Input Data.ReadOnly = False; Input Data.BitSize = 16; Input Data.DataSize = 2; Input Data.DataType = 'UINT'; Input Data.Name = 'Input Data'; Input Data.HelpString = ''; Input Data.ReadOnly = False; Input Data.BitSize = 16; Input Data.DataSize = 2; Input Data.DataType = 'UINT';
              Input Data.Name = 'Input Data'; Input Data.HelpString = ''; Input Data.ReadOnly = False; Input Data.BitSize = 16; Input Data.DataSize = 2; Input Data.DataType = 'UINT'; Input Data.Name = 'Input Data'; Input Data.HelpString = ''; Input Data.ReadOnly = False; Input Data.BitSize = 16; Input Data.DataSize = 2; Input Data.DataType = 'UINT'; Input Data.Name = 'Input Data'; Input Data.HelpString = ''; Input Data.ReadOnly = False; Input Data.BitSize = 16; Input Data.DataSize = 2; Input Data.DataType = 'UINT'; Input Data.Name = 'Input Data'; Input Data.HelpString = ''; Input Data.ReadOnly = False; Input Data.BitSize = 16; Input Data.DataSize = 2; Input Data.DataType = 'UINT'; Input Data.Name = 'Input Data'; Input Data.HelpString = ''; Input Data.ReadOnly = False; Input Data.BitSize = 16; Input Data.DataSize = 2; Input Data.DataType = 'UINT'; Input Data.Name = 'Input Data'; Input Data.HelpString = ''; Input Data.ReadOnly = False; Input Data.BitSize = 16; Input Data.DataSize = 2; Input Data.DataType = 'UINT'; Input Data.Name = 'Input Data'; Input Data.HelpString = ''; Input Data.ReadOnly = False; Input Data.BitSize = 16;
              Input Data.DataSize = 2; Input Data.DataType = 'UINT'; Input Data.Name = 'Input Data'; Input Data.HelpString = ''; Input Data.ReadOnly = False; Input Data.BitSize = 16; Input Data.DataSize = 2; Input Data.DataType = 'UINT'; Input Data.Name = 'Input Data'; Input Data.HelpString = ''; Input Data.ReadOnly = False; Input Data.BitSize = 16; Input Data.DataSize = 2; Input Data.DataType = 'UINT'; Input Data.Name = 'Input Data'; Input Data.HelpString = ''; Input Data.ReadOnly = False; Input Data.BitSize = 16; Input Data.DataSize = 2; Input Data.DataType = 'UINT'; Input Data.Name = 'Input Data'; Input Data.HelpString = ''; Input Data.ReadOnly = False; Input Data.BitSize = 16; Input Data.DataSize = 2; Input Data.DataType = 'UINT'; Input Data.Name = 'Input Data'; Input Data.HelpString = ''; Input Data.ReadOnly = False; Input Data.BitSize = 16; Input Data.DataSize = 2; Input Data.DataType = 'UINT'; Input Data.Name = 'Input Data'; Input Data.HelpString = ''; Input Data.ReadOnly = False; Input Data.BitSize = 16; Input Data.DataSize = 2; Input Data.DataType = 'UINT'; Input Data.Name = 'Input Data'; Input Data.HelpString = '';
              Input Data.ReadOnly = False; Input Data.BitSize = 16; Input Data.DataSize = 2; Input Data.DataType = 'UINT'; Input Data.Name = 'Input Data'; Input Data.HelpString = ''; Input Data.ReadOnly = False; Input Data.BitSize = 16; Input Data.DataSize = 2; Input Data.DataType = 'UINT'; Input Data.Name = 'Input Data'; Input Data.HelpString = ''; Input Data.ReadOnly = False; Input Data.BitSize = 16; Input Data.DataSize = 2; Input Data.DataType = 'UINT'; Input Data.Name = 'Input Data'; Input Data.HelpString = ''; Input Data.ReadOnly = False; Input Data.BitSize = 16; Input Data.DataSize = 2; Input Data.DataType = 'UINT'; Input Data.Name = 'Input Data'; Input Data.HelpString = ''; Input Data.ReadOnly = False; Input Data.BitSize = 16; Input Data.DataSize = 2; Input Data.DataType = 'UINT'; Input Data.Name = 'Input Data'; Input Data.HelpString = ''; Input Data.ReadOnly = False; Input Data.BitSize = 16; Input Data.DataSize = 2; Input Data.DataType = 'UINT'; Input Data.Name = 'Input Data'; Input Data.HelpString = ''; Input Data.ReadOnly = False; Input Data.BitSize = 16; Input Data.DataSize = 2; Input Data.DataType = 'UINT';
              Input Data.Name = 'Input Data'; Input Data.HelpString = ''; Input Data.ReadOnly = False; Input Data.BitSize = 16; Input Data.DataSize = 2; Input Data.DataType = 'UINT'; Input Data.Name = 'Input Data'; Input Data.HelpString = ''; Input Data.ReadOnly = False; Input Data.BitSize = 16; Input Data.DataSize = 2; Input Data.DataType = 'UINT'; Input Data.Name = 'Input Data'; Input Data.HelpString = ''; Input Data.ReadOnly = False; Input Data.BitSize = 16; Input Data.DataSize = 2; Input Data.DataType = 'UINT'; Input Data.Name = 'Input Data'; Input Data.HelpString = ''; Input Data.ReadOnly = False; Input Data.BitSize = 16; Input Data.DataSize = 2; Input Data.DataType = 'UINT'; Input Data.Name = 'Input Data'; Input Data.HelpString = ''; Input Data.ReadOnly = False; Input Data.BitSize = 16; Input Data.DataSize = 2; Input Data.DataType = 'UINT'; Input Data.Name = 'Input Data'; Input Data.HelpString = ''; Input Data.ReadOnly = False; Input Data.BitSize = 16; Input Data.DataSize = 2; Input Data.DataType = 'UINT'; Input Data.Name = 'Input Data'; Input Data.HelpString = ''; Input Data.ReadOnly = False; Input Data.BitSize = 16;
              Input Data.DataSize = 2; Input Data.DataType = 'UINT'; Input Data.Name = 'Input Data'; Input Data.HelpString = ''; Input Data.ReadOnly = False; Input Data.BitSize = 16; Input Data.DataSize = 2; Input Data.DataType = 'UINT'; Input Data.Name = 'Input Data'; Input Data.HelpString = ''; Input Data.ReadOnly = False; Input Data.BitSize = 16; Input Data.DataSize = 2; Input Data.DataType = 'UINT'; Input Data.Name = 'Input Data'; Input Data.HelpString = ''; Input Data.ReadOnly = False; Input Data.BitSize = 16; Input Data.DataSize = 2; Input Data.DataType = 'UINT'; Input Data.Name = 'Input Data'; Input Data.HelpString = ''; Input Data.ReadOnly = False; Input Data.BitSize = 16; Input Data.DataSize = 2; Input Data.DataType = 'UINT'; Input Data.Name = 'Input Data'; Input Data.HelpString = ''; Input Data.ReadOnly = False; Input Data.BitSize = 16; Input Data.DataSize = 2; Input Data.DataType = 'UINT'; Input Data.Name = 'Input Data'; Input Data.HelpString = ''; Input Data.ReadOnly = False; Input Data.BitSize = 16; Input Data.DataSize = 2; Input Data.DataType = 'UINT'; Input Data.Name = 'Input Data'; Input Data.HelpString = '';
              Input Data.ReadOnly = False; Input Data.BitSize = 16; Input Data.DataSize = 2; Input Data.DataType = 'UINT'; Input Data.Name = 'Input Data'; Input Data.HelpString = ''; Input Data.ReadOnly = False; Input Data.BitSize = 16; Input Data.DataSize = 2; Input Data.DataType = 'UINT'; Input Data.Name = 'Input Data'; Input Data.HelpString = ''; Input Data.ReadOnly = False; Input Data.BitSize = 16; Input Data.DataSize = 2; Input Data.DataType = 'UINT'; Input Data.Name = 'Input Data'; Input Data.HelpString = ''; Input Data.ReadOnly = False; Input Data.BitSize = 16; Input Data.DataSize = 2; Input Data.DataType = 'UINT'; Input Data.Name = 'Input Data'; Input Data.HelpString = ''; Input Data.ReadOnly = False; Input Data.BitSize = 16; Input Data.DataSize = 2; Input Data.DataType = 'UINT'; Input Data.Name = 'Input Data'; Input Data.HelpString = ''; Input Data.ReadOnly = False; Input Data.BitSize = 16; Input Data.DataSize = 2; Input Data.DataType = 'UINT'; Input Data.Name = 'Input Data'; Input Data.HelpString = ''; Input Data.ReadOnly = False; Input Data.BitSize = 16; Input Data.DataSize = 2; Input Data.DataType = 'UINT';
              Input Data.Name = 'Input Data'; Input Data.HelpString = ''; Input Data.ReadOnly = False; Input Data.BitSize = 16; Input Data.DataSize = 2; Input Data.DataType = 'UINT'; Input Data.Name = 'Input Data'; Input Data.HelpString = ''; Input Data.ReadOnly = False; Input Data.BitSize = 16; Input Data.DataSize = 2; Input Data.DataType = 'UINT'; Input Data.Name = 'Input Data'; Input Data.HelpString = ''; Input Data.ReadOnly = False; Input Data.BitSize = 16; Input Data.DataSize = 2; Input Data.DataType = 'UINT'; Input Data.Name = 'Input Data'; Input Data.HelpString = ''; Input Data.ReadOnly = False; Input Data.BitSize = 16; Input Data.DataSize = 2; Input Data.DataType = 'UINT'; Input Data.Name = 'Input Data'; Input Data.HelpString = ''; Input Data.ReadOnly = False; Input Data.BitSize = 16; Input Data.DataSize = 2; Input Data.DataType = 'UINT'; Input Data.Name = 'Input Data'; Input Data.HelpString = ''; Input Data.ReadOnly = False; Input Data.BitSize = 16; Input Data.DataSize = 2; Input Data.DataType = 'UINT'; Input Data.Name = 'Input Data'; Input Data.HelpString = ''; Input Data.ReadOnly = False; Input Data.BitSize = 16;
              Input Data.DataSize = 2; Input Data.DataType = 'UINT'; Input Data.Name = 'Input Data'; Input Data.HelpString = ''; Input Data.ReadOnly = False; Input Data.BitSize = 16; Input Data.DataSize = 2; Input Data.DataType = 'UINT'; Input Data.Name = 'Input Data'; Input Data.HelpString = ''; Input Data.ReadOnly = False; Input Data.BitSize = 16; Input Data.DataSize = 2; Input Data.DataType = 'UINT'; Input Data.Name = 'Input Data'; Input Data.HelpString = ''; Input Data.ReadOnly = False; Input Data.BitSize = 16; Input Data.DataSize = 2; Input Data.DataType = 'UINT'; Input Data.Name = 'Input Data'; Input Data.HelpString = ''; Input Data.ReadOnly = False; Input Data.BitSize = 16; Input Data.DataSize = 2; Input Data.DataType = 'UINT'; Input Data.Name = 'Input Data'; Input Data.HelpString = ''; Input Data.ReadOnly = False; Input Data.BitSize = 16; Input Data.DataSize = 2; Input Data.DataType = 'UINT'; Input Data.Name = 'Input Data'; Input Data.HelpString = ''; Input Data.ReadOnly = False; Input Data.BitSize = 16; Input Data.DataSize = 2; Input Data.DataType = 'UINT'; Input Data.Name = 'Input Data'; Input Data.HelpString = '';
              Input Data.ReadOnly = False; Input Data.BitSize = 16; Input Data.DataSize = 2; Input Data.DataType = 'UINT'; Input Data.Name = 'Input Data'; Input Data.HelpString = ''; Input Data.ReadOnly = False; Input Data.BitSize = 16; Input Data.DataSize = 2; Input Data.DataType = 'UINT'; Input Data.Name = 'Input Data'; Input Data.HelpString = ''; Input Data.ReadOnly = False; Input Data.BitSize = 16; Input Data.DataSize = 2; Input Data.DataType = 'UINT'; Input Data.Name = 'Input Data'; Input Data.HelpString = ''; Input Data.ReadOnly = False; Input Data.BitSize = 16; Input Data.DataSize = 2; Input Data.DataType = 'UINT'; Input Data.Name = 'Input Data'; Input Data.HelpString = ''; Input Data.ReadOnly = False; Input Data.BitSize = 16; Input Data.DataSize = 2; Input Data.DataType = 'UINT'; Input Data.Name = 'Input Data'; Input Data.HelpString = ''; Input Data.ReadOnly = False; Input Data.BitSize = 16; Input Data.DataSize = 2; Input Data.DataType = 'UINT'; Input Data.Name = 'Input Data'; Input Data.HelpString = ''; Input Data.ReadOnly = False; Input Data.BitSize = 16; Input Data.DataSize = 2; Input Data.DataType = 'UINT';
              Input Data.Name = 'Input Data'; Input Data.HelpString = ''; Input Data.ReadOnly = False; Input Data.BitSize = 16; Input Data.DataSize = 2; Input Data.DataType = 'UINT'; Input Data.Name = 'Input Data'; Input Data.HelpString = ''; Input Data.ReadOnly = False; Input Data.BitSize = 16; Input Data.DataSize = 2; Input Data.DataType = 'UINT'; Input Data.Name = 'Input Data'; Input Data.HelpString = ''; Input Data.ReadOnly = False; Input Data.BitSize = 16; Input Data.DataSize = 2; Input Data.DataType = 'UINT'; Input Data.Name = 'Input Data'; Input Data.HelpString = ''; Input Data.ReadOnly = False; Input Data.BitSize = 16; Input Data.DataSize = 2; Input Data.DataType = 'UINT'; Input Data.Name = 'Input Data'; Input Data.HelpString = ''; Input Data.ReadOnly = False; Input Data.BitSize = 16; Input Data.DataSize = 2; Input Data.DataType = 'UINT'; Input Data.Name = 'Input Data'; Input Data.HelpString = ''; Input Data.ReadOnly = False; Input Data.BitSize = 16; Input Data.DataSize = 2; Input Data.DataType = 'UINT'; Input Data.Name = 'Input Data'; Input Data.HelpString = ''; Input Data.ReadOnly = False; Input Data.BitSize = 16;
              Input Data.DataSize = 2; Input Data.DataType = 'UINT'; Input Data.Name = 'Input Data'; Input Data.HelpString = ''; Input Data.ReadOnly = False; Input Data.BitSize = 16; Input Data.DataSize = 2; Input Data.DataType = 'UINT'; Input Data.Name = 'Input Data'; Input Data.HelpString = ''; Input Data.ReadOnly = False; Input Data.BitSize = 16; Input Data.DataSize = 2; Input Data.DataType = 'UINT'; Input Data.Name = 'Input Data'; Input Data.HelpString = ''; Input Data.ReadOnly = False; Input Data.BitSize = 16; Input Data.DataSize = 2; Input Data.DataType = 'UINT'; Input Data.Name = 'Input Data'; Input Data.HelpString = ''; Input Data.ReadOnly = False; Input Data.BitSize = 16; Input Data.DataSize = 2; Input Data.DataType = 'UINT'; Input Data.Name = 'Input Data'; Input Data.HelpString = ''; Input Data.ReadOnly = False; Input Data.BitSize = 16; Input Data.DataSize = 2; Input Data.DataType = 'UINT'; Input Data.Name = 'Input Data'; Input Data.HelpString = ''; Input Data.ReadOnly = False; Input Data.BitSize = 16; Input Data.DataSize = 2; Input Data.DataType = 'UINT'; Input Data.Name = 'Input Data'; Input Data.HelpString = '';
              Input Data.ReadOnly = False; Input Data.BitSize = 16; Input Data.DataSize = 2; Input Data.DataType = 'UINT'; Input Data.Name = 'Input Data'; Input Data.HelpString = ''; Input Data.ReadOnly = False; Input Data.BitSize = 16; Input Data.DataSize = 2; Input Data.DataType = 'UINT'; Input Data.Name = 'Input Data'; Input Data.HelpString = ''; Input Data.ReadOnly = False; Input Data.BitSize = 16; Input Data.DataSize = 2; Input Data.DataType = 'UINT'; Input Data.Name = 'Input Data'; Input Data.HelpString = ''; Input Data.ReadOnly = False; Input Data.BitSize = 16; Input Data.DataSize = 2; Input Data.DataType = 'UINT'; Input Data.Name = 'Input Data'; Input Data.HelpString = ''; Input Data.ReadOnly = False; Input Data.BitSize = 16; Input Data.DataSize = 2; Input Data.DataType = 'UINT'; Input Data.Name = 'Input Data'; Input Data.HelpString = ''; Input Data.ReadOnly = False; Input Data.BitSize = 16; Input Data.DataSize = 2; Input Data.DataType = 'UINT'; Input Data.Name = 'Input Data'; Input Data.HelpString = ''; Input Data.ReadOnly = False; Input Data.BitSize = 16; Input Data.DataSize = 2; Input Data.DataType = 'UINT';
              Input Data.Name = 'Input Data'; Input Data.HelpString = ''; Input Data.ReadOnly = False; Input Data.BitSize = 16; Input Data.DataSize = 2; Input Data.DataType = 'UINT'; Input Data.Name = 'Input Data'; Input Data.HelpString = ''; Input Data.ReadOnly = False; Input Data.BitSize = 16; Input Data.DataSize = 2; Input Data.DataType = 'UINT'; Input Data.Name = 'Input Data'; Input Data.HelpString = ''; Input Data.ReadOnly = False; Input Data.BitSize = 16; Input Data.DataSize = 2; Input Data.DataType = 'UINT'; Input Data.Name = 'Input Data'; Input Data.HelpString = ''; Input Data.ReadOnly = False; Input Data.BitSize = 16; Input Data.DataSize = 2; Input Data.DataType = 'UINT'; Input Data.Name = 'Input Data'; Input Data.HelpString = ''; Input Data.ReadOnly = False; Input Data.BitSize = 16; Input Data.DataSize = 2; Input Data.DataType = 'UINT'; Input Data.Name = 'Input Data'; Input Data.HelpString = ''; Input Data.ReadOnly = False; Input Data.BitSize = 16; Input Data.DataSize = 2; Input Data.DataType = 'UINT'; Input Data.Name = 'Input Data'; Input Data.HelpString = ''; Input Data.ReadOnly = False; Input Data.BitSize = 16;
              Input Data.DataSize = 2; Input Data.DataType = 'UINT'; Input Data.Name = 'Input Data'; Input Data.HelpString = ''; Input Data.ReadOnly = False; Input Data.BitSize = 16; Input Data.DataSize = 2; Input Data.DataType = 'UINT'; Input Data.Name = 'Input Data'; Input Data.HelpString = ''; Input Data.ReadOnly = False; Input Data.BitSize = 16; Input Data.DataSize = 2; Input Data.DataType = 'UINT'; Input Data.Name = 'Input Data'; Input Data.HelpString = ''; Input Data.ReadOnly = False; Input Data.BitSize = 16; Input Data.DataSize = 2; Input Data.DataType = 'UINT'; Input Data.Name = 'Input Data'; Input Data.HelpString = ''; Input Data.ReadOnly = False; Input Data.BitSize = 16; Input Data.DataSize = 2; Input Data.DataType = 'UINT'; Input Data.Name = 'Input Data'; Input Data.HelpString = ''; Input Data.ReadOnly = False; Input Data.BitSize = 16; Input Data.DataSize = 2; Input Data.DataType = 'UINT'; Input Data.Name = 'Input Data'; Input Data.HelpString = ''; Input Data.ReadOnly = False; Input Data.BitSize = 16; Input Data.DataSize = 2; Input Data.DataType = 'UINT'; Input Data.Name = 'Input Data'; Input Data.HelpString = '';
              Input Data.ReadOnly = False; Input Data.BitSize = 16; Input Data.DataSize = 2; Input Data.DataType = 'UINT'; Input Data.Name = 'Input Data'; Input Data.HelpString = ''; Input Data.ReadOnly = False; Input Data.BitSize = 16; Input Data.DataSize = 2; Input Data.DataType = 'UINT'; Input Data.Name = 'Input Data'; Input Data.HelpString = ''; Input Data.ReadOnly = False; Input Data.BitSize = 16; Input Data.DataSize = 2; Input Data.DataType = 'UINT'; Input Data.Name = 'Input Data'; Input Data.HelpString = ''; Input Data.ReadOnly = False; Input Data.BitSize = 16; Input Data.DataSize = 2; Input Data.DataType = 'UINT'; Input Data.Name = 'Input Data'; Input Data.HelpString = ''; Input Data.ReadOnly = False; Input Data.BitSize = 16; Input Data.DataSize = 2; Input Data.DataType = 'UINT'; Input Data.Name = 'Input Data'; Input Data.HelpString = ''; Input Data.ReadOnly = False; Input Data.BitSize = 16; Input Data.DataSize = 2; Input Data.DataType = 'UINT'; Input Data.Name = 'Input Data'; Input Data.HelpString = ''; Input Data.ReadOnly = False; Input Data.BitSize = 16; Input Data.DataSize = 2; Input Data.DataType = 'UINT';
              Input Data.Name = 'Input Data'; Input Data.HelpString = ''; Input Data.ReadOnly = False; Input Data.BitSize = 16; Input Data.DataSize = 2; Input Data.DataType = 'UINT'; Input Data.Name = 'Input Data'; Input Data.HelpString = ''; Input Data.ReadOnly = False; Input Data.BitSize = 16; Input Data.DataSize = 2; Input Data.DataType = 'UINT'; Input Data.Name = 'Input Data'; Input Data.HelpString = ''; Input Data.ReadOnly = False; Input Data.BitSize = 16; Input Data.DataSize = 2; Input Data.DataType = 'UINT'; Input Data.Name = 'Input Data'; Input Data.HelpString = ''; Input Data.ReadOnly = False; Input Data.BitSize = 16; Input Data.DataSize = 2; Input Data.DataType = 'UINT'; Input Data.Name = 'Input Data'; Input Data.HelpString = ''; Input Data.ReadOnly = False; Input Data.BitSize = 16; Input Data.DataSize = 2; Input Data.DataType = 'UINT'; Input Data.Name = 'Input Data'; Input Data.HelpString = ''; Input Data.ReadOnly = False; Input Data.BitSize = 16; Input Data.DataSize = 2; Input Data.DataType = 'UINT'; Input Data.Name = 'Input Data'; Input Data.HelpString = ''; Input Data.ReadOnly = False; Input Data.BitSize = 16;
              Input Data.DataSize = 2; Input Data.DataType = 'UINT'; Input Data.Name = 'Input Data'; Input Data.HelpString = ''; Input Data.ReadOnly = False; Input Data.BitSize = 16; Input Data.DataSize = 2; Input Data.DataType = 'UINT'; Input Data.Name = 'Input Data'; Input Data.HelpString = ''; Input Data.ReadOnly = False; Input Data.BitSize = 16; Input Data.DataSize = 2; Input Data.DataType = 'UINT'; Input Data.Name = 'Input Data'; Input Data.HelpString = ''; Input Data.ReadOnly = False; Input Data.BitSize = 16; Input Data.DataSize = 2; Input Data.DataType = 'UINT'; Input Data.Name = 'Input Data'; Input Data.HelpString = ''; Input Data.ReadOnly = False; Input Data.BitSize = 16; Input Data.DataSize = 2; Input Data.DataType = 'UINT'; Input Data.Name = 'Input Data'; Input Data.HelpString = ''; Input Data.ReadOnly = False; Input Data.BitSize = 16; Input Data.DataSize = 2; Input Data.DataType = 'UINT'; Input Data.Name = 'Input Data'; Input Data.HelpString = ''; Input Data.ReadOnly = False; Input Data.BitSize = 16; Input Data.DataSize = 2; Input Data.DataType = 'UINT'; Input Data.Name = 'Input Data'; Input Data.HelpString = '';
              Input Data.ReadOnly = False; Input Data.BitSize = 16; Input Data.DataSize = 2; Input Data.DataType = 'UINT'; Input Data.Name = 'Input Data'; Input Data.HelpString = ''; Input Data.ReadOnly = False; Input Data.BitSize = 16; Input Data.DataSize = 2; Input Data.DataType = 'UINT'; Input Data.Name = 'Input Data'; Input Data.HelpString = ''; Input Data.ReadOnly = False; Input Data.BitSize = 16; Input Data.DataSize = 2; Input Data.DataType = 'UINT'; Input Data.Name = 'Input Data'; Input Data.HelpString = ''; Input Data.ReadOnly = False; Input Data.BitSize = 16; Input Data.DataSize = 2; Input Data.DataType = 'UINT'; Input Data.Name = 'Input Data'; Input Data.HelpString = ''; Input Data.ReadOnly = False; Input Data.BitSize = 16; Input Data.DataSize = 2; Input Data.DataType = 'UINT'; Input Data.Name = 'Input Data'; Input Data.HelpString = ''; Input Data.ReadOnly = False; Input Data.BitSize = 16; Input Data.DataSize = 2; Input Data.DataType = 'UINT'; Input Data.Name = 'Input Data'; Input Data.HelpString = ''; Input Data.ReadOnly = False; Input Data.BitSize = 16; Input Data.DataSize = 2; Input Data.DataType = 'UINT';
              Input Data.Name = 'Input Data'; Input Data.HelpString = ''; Input Data.ReadOnly = False; Input Data.BitSize = 16; Input Data.DataSize = 2; Input Data.DataType = 'UINT'; Input Data.Name = 'Input Data'; Input Data.HelpString = ''; Input Data.ReadOnly = False; Input Data.BitSize = 16; Input Data.DataSize = 2; Input Data.DataType = 'UINT'; Input Data.Name = 'Input Data'; Input Data.HelpString = ''; Input Data.ReadOnly = False; Input Data.BitSize = 16; Input Data.DataSize = 2; Input Data.DataType = 'UINT'; Input Data.Name = 'Input Data'; Input Data.HelpString = ''; Input Data.ReadOnly = False; Input Data.BitSize = 16; Input Data.DataSize = 2; Input Data.DataType = 'UINT'; Input Data.Name = 'Input Data'; Input Data.HelpString = ''; Input Data.ReadOnly = False; Input Data.BitSize = 16; Input Data.DataSize = 2; Input Data.DataType = 'UINT'; Input Data.Name = 'Input Data'; Input Data.HelpString = ''; Input Data.ReadOnly = False; Input Data.BitSize = 16; Input Data.DataSize = 2; Input Data.DataType = 'UINT'; Input Data.Name = 'Input Data'; Input Data.HelpString = ''; Input Data.ReadOnly = False; Input Data.BitSize = 16;
              Input Data.DataSize = 2; Input Data.DataType = 'UINT'; Input Data.Name = 'Input Data'; Input Data.HelpString = ''; Input Data.ReadOnly = False; Input Data.BitSize = 16; Input Data.DataSize = 2; Input Data.DataType = 'UINT'; Input Data.Name = 'Input Data'; Input Data.HelpString = ''; Input Data.ReadOnly = False; Input Data.BitSize = 16; Input Data.DataSize = 2; Input Data.DataType = 'UINT'; Input Data.Name = 'Input Data'; Input Data.HelpString = ''; Input Data.ReadOnly = False; Input Data.BitSize = 16; Input Data.DataSize = 2; Input Data.DataType = 'UINT'; Input Data.Name = 'Input Data'; Input Data.HelpString = ''; Input Data.ReadOnly = False; Input Data.BitSize = 16; Input Data.DataSize = 2; Input Data.DataType = 'UINT'; Input Data.Name = 'Input Data'; Input Data.HelpString = ''; Input Data.ReadOnly = False; Input Data.BitSize = 16; Input Data.DataSize = 2; Input Data.DataType = 'UINT'; Input Data.Name = 'Input Data'; Input Data.HelpString = ''; Input Data.ReadOnly = False; Input Data.BitSize = 16; Input Data.DataSize = 2; Input Data.DataType = 'UINT'; Input Data.Name = 'Input Data'; Input Data.HelpString = '';
              Input Data.ReadOnly = False; Input Data.BitSize = 16; Input Data.DataSize = 2; Input Data.DataType = 'UINT'; Input Data.Name = 'Input Data'; Input Data.HelpString = ''; Input Data.ReadOnly = False; Input Data.BitSize = 16; Input Data.DataSize = 2; Input Data.DataType = 'UINT'; Input Data.Name = 'Input Data'; Input Data.HelpString = ''; Input Data.ReadOnly = False; Input Data.BitSize = 16; Input Data.DataSize = 2; Input Data.DataType = 'UINT'; Input Data.Name = 'Input Data'; Input Data.HelpString = ''; Input Data.ReadOnly = False; Input Data.BitSize = 16; Input Data.DataSize = 2; Input Data.DataType = 'UINT'; Input Data.Name = 'Input Data'; Input Data.HelpString = ''; Input Data.ReadOnly = False; Input Data.BitSize = 16; Input Data.DataSize = 2; Input Data.DataType = 'UINT'; Input Data.Name = 'Input Data'; Input Data.HelpString = ''; Input Data.ReadOnly = False; Input Data.BitSize = 16; Input Data.DataSize = 2; Input Data.DataType = 'UINT'; Input Data.Name = 'Input Data'; Input Data.HelpString = ''; Input Data.ReadOnly = False; Input Data.BitSize = 16; Input Data.DataSize = 2; Input Data.DataType = 'UINT';
              Input Data.Name = 'Input Data'; Input Data.HelpString = ''; Input Data.ReadOnly = False; Input Data.BitSize = 16; Input Data.DataSize = 2; Input Data.DataType = 'UINT'; Input Data.Name = 'Input Data'; Input Data.HelpString = ''; Input Data.ReadOnly = False; Input Data.BitSize = 16; Input Data.DataSize = 2; Input Data.DataType = 'UINT'; Input Data.Name = 'Input Data'; Input Data.HelpString = ''; Input Data.ReadOnly = False; Input Data.BitSize = 16; Input Data.DataSize = 2; Input Data.DataType = 'UINT'; Input Data.Name = 'Input Data'; Input Data.HelpString = ''; Input Data.ReadOnly = False; Input Data.BitSize = 16; Input Data.DataSize = 2; Input Data.DataType = 'UINT'; Input Data.Name = 'Input Data'; Input Data.HelpString = ''; Input Data.ReadOnly = False; Input Data.BitSize = 16; Input Data.DataSize = 2; Input Data.DataType = 'UINT'; Input Data.Name = 'Input Data'; Input Data.HelpString = ''; Input Data.ReadOnly = False; Input Data.BitSize = 16; Input Data.DataSize = 2; Input Data.DataType = 'UINT'; Input Data.Name = 'Input Data'; Input Data.HelpString = ''; Input Data.ReadOnly = False; Input Data.BitSize = 16;
              Input Data.DataSize = 2; Input Data.DataType = 'UINT'; Input Data.Name = 'Input Data'; Input Data.HelpString = ''; Input Data.ReadOnly = False; Input Data.BitSize = 16; Input Data.DataSize = 2; Input Data.DataType = 'UINT'; Input Data.Name = 'Input Data'; Input Data.HelpString = ''; Input Data.ReadOnly = False; Input Data.BitSize = 16; Input Data.DataSize = 2; Input Data.DataType = 'UINT'; Input Data.Name = 'Input Data'; Input Data.HelpString = ''; Input Data.ReadOnly = False; Input Data.BitSize = 16; Input Data.DataSize = 2; Input Data.DataType = 'UINT'; Input Data.Name = 'Input Data'; Input Data.HelpString = ''; Input Data.ReadOnly = False; Input Data.BitSize = 16; Input Data.DataSize = 2; Input Data.DataType = 'UINT'; Input Data.Name = 'Input Data'; Input Data.HelpString = ''; Input Data.ReadOnly = False; Input Data.BitSize = 16; Input Data.DataSize = 2; Input Data.DataType = 'UINT'; Input Data.Name = 'Input Data'; Input Data.HelpString = ''; Input Data.ReadOnly = False; Input Data.BitSize = 16; Input Data.DataSize = 2; Input Data.DataType = 'UINT'; Input Data.Name = 'Input Data'; Input Data.HelpString = '';
              Input Data.ReadOnly = False; Input Data.BitSize = 16; Input Data.DataSize = 2; Input Data.DataType = 'UINT'; Input Data.Name = 'Input Data'; Input Data.HelpString = ''; Input Data.ReadOnly = False; Input Data.BitSize = 16; Input Data.DataSize = 2; Input Data.DataType = 'UINT'; Input Data.Name = 'Input Data'; Input Data.HelpString = ''; Input Data.ReadOnly = False; Input Data.BitSize = 16; Input Data.DataSize = 2; Input Data.DataType = 'UINT'; Input Data.Name = 'Input Data'; Input Data.HelpString = ''; Input Data.ReadOnly = False; Input Data.BitSize = 16; Input Data.DataSize = 2; Input Data.DataType = 'UINT'; Input Data.Name = 'Input Data'; Input Data.HelpString = ''; Input Data.ReadOnly = False; Input Data.BitSize = 16; Input Data.DataSize = 2; Input Data.DataType = 'UINT'; Input Data.Name = 'Input Data'; Input Data.HelpString = ''; Input Data.ReadOnly = False; Input Data.BitSize = 16; Input Data.DataSize = 2; Input Data.DataType = 'UINT'; Input Data.Name = 'Input Data'; Input Data.HelpString = ''; Input Data.ReadOnly = False; Input Data.BitSize = 16; Input Data.DataSize = 2; Input Data.DataType = 'UINT';
              Input Data.Name = 'Input Data'; Input Data.HelpString = ''; Input Data.ReadOnly = False; Input Data.BitSize = 16; Input Data.DataSize = 2; Input Data.DataType = 'UINT'; Input Data.Name = 'Input Data'; Input Data.HelpString = ''; Input Data.ReadOnly = False; Input Data.BitSize = 16; Input Data.DataSize = 2; Input Data.DataType = 'UINT'; Input Data.Name = 'Input Data'; Input Data.HelpString = ''; Input Data.ReadOnly = False; Input Data.BitSize = 16; Input Data.DataSize = 2; Input Data.DataType = 'UINT'; Input Data.Name = 'Input Data'; Input Data.HelpString = ''; Input Data.ReadOnly = False; Input Data.BitSize = 16; Input Data.DataSize = 2; Input Data.DataType = 'UINT'; Input Data.Name = 'Input Data'; Input Data.HelpString = ''; Input Data.ReadOnly = False; Input Data.BitSize = 16; Input Data.DataSize = 2; Input Data.DataType = 'UINT'; Input Data.Name = 'Input Data'; Input Data.HelpString = ''; Input Data.ReadOnly = False; Input Data.BitSize = 16; Input Data.DataSize = 2; Input Data.DataType = 'UINT'; Input Data.Name = 'Input Data'; Input Data.HelpString = ''; Input Data.ReadOnly = False; Input Data.BitSize = 16;
              Input Data.DataSize = 2; Input Data.DataType = 'UINT'; Input Data.Name = 'Input Data'; Input Data.HelpString = ''; Input Data.ReadOnly = False; Input Data.BitSize = 16; Input Data.DataSize = 2; Input Data.DataType = 'UINT'; Input Data.Name = 'Input Data'; Input Data.HelpString = ''; Input Data.ReadOnly = False; Input Data.BitSize = 16; Input Data.DataSize = 2; Input Data.DataType = 'UINT'; Input Data.Name = 'Input Data'; Input Data.HelpString = ''; Input Data.ReadOnly = False; Input Data.BitSize = 16; Input Data.DataSize = 2; Input Data.DataType = 'UINT'; Input Data.Name = 'Input Data'; Input Data.HelpString = ''; Input Data.ReadOnly = False; Input Data.BitSize = 16; Input Data.DataSize = 2; Input Data.DataType = 'UINT'; Input Data.Name = 'Input Data'; Input Data.HelpString = ''; Input Data.ReadOnly = False; Input Data.BitSize = 16; Input Data.DataSize = 2; Input Data.DataType = 'UINT'; Input Data.Name = 'Input Data'; Input Data.HelpString = ''; Input Data.ReadOnly = False; Input Data.BitSize = 16; Input Data.DataSize = 2; Input Data.DataType = 'UINT'; Input Data.Name = 'Input Data'; Input Data.HelpString = '';
              Input Data.ReadOnly = False; Input Data.BitSize = 16; Input Data.DataSize = 2; Input Data.DataType = 'UINT'; Input Data.Name = 'Input Data'; Input Data.HelpString = ''; Input Data.ReadOnly = False; Input Data.BitSize = 16; Input Data.DataSize = 2; Input Data.DataType = 'UINT'; Input Data.Name = 'Input Data'; Input Data.HelpString = ''; Input Data.ReadOnly = False; Input Data.BitSize = 16; Input Data.DataSize = 2; Input Data.DataType = 'UINT'; Input Data.Name = 'Input Data'; Input Data.HelpString = ''; Input Data.ReadOnly = False; Input Data.BitSize = 16; Input Data.DataSize = 2; Input Data.DataType = 'UINT'; Input Data.Name = 'Input Data'; Input Data.HelpString = ''; Input Data.ReadOnly = False; Input Data.BitSize = 16; Input Data.DataSize = 2; Input Data.DataType = 'UINT'; Input Data.Name = 'Input Data'; Input Data.HelpString = ''; Input Data.ReadOnly = False; Input Data.BitSize = 16; Input Data.DataSize = 2; Input Data.DataType = 'UINT'; Input Data.Name = 'Input Data'; Input Data.HelpString = ''; Input Data.ReadOnly = False; Input Data.BitSize = 16; Input Data.DataSize = 2; Input Data.DataType = 'UINT';
              Input Data.Name = 'Input Data'; Input Data.HelpString = ''; Input Data.ReadOnly = False; Input Data.BitSize = 16; Input Data.DataSize = 2; Input Data.DataType = 'UINT'; Input Data.Name = 'Input Data'; Input Data.HelpString = ''; Input Data.ReadOnly = False; Input Data.BitSize = 16; Input Data.DataSize = 2; Input Data.DataType = 'UINT'; Input Data.Name = 'Input Data'; Input Data.HelpString = ''; Input Data.ReadOnly = False; Input Data.BitSize = 16; Input Data.DataSize = 2; Input Data.DataType = 'UINT'; Input Data.Name = 'Input Data'; Input Data.HelpString = ''; Input Data.ReadOnly = False; Input Data.BitSize = 16; Input Data.DataSize = 2; Input Data.DataType = 'UINT'; Input Data.Name = 'Input Data'; Input Data.HelpString = ''; Input Data.ReadOnly = False; Input Data.BitSize = 16; Input Data.DataSize = 2; Input Data.DataType = 'UINT'; Input Data.Name = 'Input Data'; Input Data.HelpString = ''; Input Data.ReadOnly = False; Input Data.BitSize = 16; Input Data.DataSize = 2; Input Data.DataType = 'UINT'; Input Data.Name = 'Input Data'; Input Data.HelpString = ''; Input Data.ReadOnly = False; Input Data.BitSize = 16;
              Input Data.DataSize = 2; Input Data.DataType = 'UINT'; Input Data.Name = 'Input Data'; Input Data.HelpString = ''; Input Data.ReadOnly = False; Input Data.BitSize = 16; Input Data.DataSize = 2; Input Data.DataType = 'UINT'; Input Data.Name = 'Input Data'; Input Data.HelpString = ''; Input Data.ReadOnly = False; Input Data.BitSize = 16; Input Data.DataSize = 2; Input Data.DataType = 'UINT'; Input Data.Name = 'Input Data'; Input Data.HelpString = ''; Input Data.ReadOnly = False; Input Data.BitSize = 16; Input Data.DataSize = 2; Input Data.DataType = 'UINT'; Input Data.Name = 'Input Data'; Input Data.HelpString = ''; Input Data.ReadOnly = False; Input Data.BitSize = 16; Input Data.DataSize = 2; Input Data.DataType = 'UINT'; Input Data.Name = 'Input Data'; Input Data.HelpString = ''; Input Data.ReadOnly = False; Input Data.BitSize = 16; Input Data.DataSize = 2; Input Data.DataType = 'UINT'; Input Data.Name = 'Input Data'; Input Data.HelpString = ''; Input Data.ReadOnly = False; Input Data.BitSize = 16; Input Data.DataSize = 2; Input Data.DataType = 'UINT'; Input Data.Name = 'Input Data'; Input Data.HelpString = '';
              Input Data.ReadOnly = False; Input Data.BitSize = 16; Input Data.DataSize = 2; Input Data.DataType = 'UINT'; Input Data.Name = 'Input Data'; Input Data.HelpString = ''; Input Data.ReadOnly = False; Input Data.BitSize = 16; Input Data.DataSize = 2; Input Data.DataType = 'UINT'; Input Data.Name = 'Input Data'; Input Data.HelpString = ''; Input Data.ReadOnly = False; Input Data.BitSize = 16; Input Data.DataSize = 2; Input Data.DataType = 'UINT'; Input Data.Name = 'Input Data'; Input Data.HelpString = ''; Input Data.ReadOnly = False; Input Data.BitSize = 16; Input Data.DataSize = 2; Input Data.DataType = 'UINT'; Input Data.Name = 'Input Data'; Input Data.HelpString = ''; Input Data.ReadOnly = False; Input Data.BitSize = 16; Input Data.DataSize = 2; Input Data.DataType = 'UINT'; Input Data.Name = 'Input Data'; Input Data.HelpString = ''; Input Data.ReadOnly = False; Input Data.BitSize = 16; Input Data.DataSize = 2; Input Data.DataType = 'UINT'; Output Data.Name = 'Output Data'; Output Data.HelpString = ''; Output Data.ReadOnly = False; Output Data.BitSize = 16; Output Data.DataSize = 2; Output Data.DataType = 'UINT';
              Output Data.Name = 'Output Data'; Output Data.HelpString = ''; Output Data.ReadOnly = False; Output Data.BitSize = 16; Output Data.DataSize = 2; Output Data.DataType = 'UINT'; Output Data.Name = 'Output Data'; Output Data.HelpString = ''; Output Data.ReadOnly = False; Output Data.BitSize = 16; Output Data.DataSize = 2; Output Data.DataType = 'UINT'; Output Data.Name = 'Output Data'; Output Data.HelpString = ''; Output Data.ReadOnly = False; Output Data.BitSize = 16; Output Data.DataSize = 2; Output Data.DataType = 'UINT'; Output Data.Name = 'Output Data'; Output Data.HelpString = ''; Output Data.ReadOnly = False; Output Data.BitSize = 16; Output Data.DataSize = 2; Output Data.DataType = 'UINT'; Output Data.Name = 'Output Data'; Output Data.HelpString = ''; Output Data.ReadOnly = False; Output Data.BitSize = 16; Output Data.DataSize = 2; Output Data.DataType = 'UINT'; Output Data.Name = 'Output Data'; Output Data.HelpString = ''; Output Data.ReadOnly = False; Output Data.BitSize = 16; Output Data.DataSize = 2; Output Data.DataType = 'UINT'; Output Data.Name = 'Output Data'; Output Data.HelpString = ''; Output Data.ReadOnly = False; Output Data.BitSize = 16;
              Output Data.DataSize = 2; Output Data.DataType = 'UINT'; Output Data.Name = 'Output Data'; Output Data.HelpString = ''; Output Data.ReadOnly = False; Output Data.BitSize = 16; Output Data.DataSize = 2; Output Data.DataType = 'UINT'; Output Data.Name = 'Output Data'; Output Data.HelpString = ''; Output Data.ReadOnly = False; Output Data.BitSize = 16; Output Data.DataSize = 2; Output Data.DataType = 'UINT'; Output Data.Name = 'Output Data'; Output Data.HelpString = ''; Output Data.ReadOnly = False; Output Data.BitSize = 16; Output Data.DataSize = 2; Output Data.DataType = 'UINT'; Output Data.Name = 'Output Data'; Output Data.HelpString = ''; Output Data.ReadOnly = False; Output Data.BitSize = 16; Output Data.DataSize = 2; Output Data.DataType = 'UINT'; Output Data.Name = 'Output Data'; Output Data.HelpString = ''; Output Data.ReadOnly = False; Output Data.BitSize = 16; Output Data.DataSize = 2; Output Data.DataType = 'UINT'; Output Data.Name = 'Output Data'; Output Data.HelpString = ''; Output Data.ReadOnly = False; Output Data.BitSize = 16; Output Data.DataSize = 2; Output Data.DataType = 'UINT'; Output Data.Name = 'Output Data'; Output Data.HelpString = '';
              Output Data.ReadOnly = False; Output Data.BitSize = 16; Output Data.DataSize = 2; Output Data.DataType = 'UINT'; Output Data.Name = 'Output Data'; Output Data.HelpString = ''; Output Data.ReadOnly = False; Output Data.BitSize = 16; Output Data.DataSize = 2; Output Data.DataType = 'UINT'; Output Data.Name = 'Output Data'; Output Data.HelpString = ''; Output Data.ReadOnly = False; Output Data.BitSize = 16; Output Data.DataSize = 2; Output Data.DataType = 'UINT'; Output Data.Name = 'Output Data'; Output Data.HelpString = ''; Output Data.ReadOnly = False; Output Data.BitSize = 16; Output Data.DataSize = 2; Output Data.DataType = 'UINT'; Output Data.Name = 'Output Data'; Output Data.HelpString = ''; Output Data.ReadOnly = False; Output Data.BitSize = 16; Output Data.DataSize = 2; Output Data.DataType = 'UINT'; Output Data.Name = 'Output Data'; Output Data.HelpString = ''; Output Data.ReadOnly = False; Output Data.BitSize = 16; Output Data.DataSize = 2; Output Data.DataType = 'UINT'; Output Data.Name = 'Output Data'; Output Data.HelpString = ''; Output Data.ReadOnly = False; Output Data.BitSize = 16; Output Data.DataSize = 2; Output Data.DataType = 'UINT';
              Output Data.Name = 'Output Data'; Output Data.HelpString = ''; Output Data.ReadOnly = False; Output Data.BitSize = 16; Output Data.DataSize = 2; Output Data.DataType = 'UINT'; Output Data.Name = 'Output Data'; Output Data.HelpString = ''; Output Data.ReadOnly = False; Output Data.BitSize = 16; Output Data.DataSize = 2; Output Data.DataType = 'UINT'; Output Data.Name = 'Output Data'; Output Data.HelpString = ''; Output Data.ReadOnly = False; Output Data.BitSize = 16; Output Data.DataSize = 2; Output Data.DataType = 'UINT'; Output Data.Name = 'Output Data'; Output Data.HelpString = ''; Output Data.ReadOnly = False; Output Data.BitSize = 16; Output Data.DataSize = 2; Output Data.DataType = 'UINT'; Output Data.Name = 'Output Data'; Output Data.HelpString = ''; Output Data.ReadOnly = False; Output Data.BitSize = 16; Output Data.DataSize = 2; Output Data.DataType = 'UINT'; Output Data.Name = 'Output Data'; Output Data.HelpString = ''; Output Data.ReadOnly = False; Output Data.BitSize = 16; Output Data.DataSize = 2; Output Data.DataType = 'UINT'; Output Data.Name = 'Output Data'; Output Data.HelpString = ''; Output Data.ReadOnly = False; Output Data.BitSize = 16;
              Output Data.DataSize = 2; Output Data.DataType = 'UINT'; Output Data.Name = 'Output Data'; Output Data.HelpString = ''; Output Data.ReadOnly = False; Output Data.BitSize = 16; Output Data.DataSize = 2; Output Data.DataType = 'UINT'; Output Data.Name = 'Output Data'; Output Data.HelpString = ''; Output Data.ReadOnly = False; Output Data.BitSize = 16; Output Data.DataSize = 2; Output Data.DataType = 'UINT'; Output Data.Name = 'Output Data'; Output Data.HelpString = ''; Output Data.ReadOnly = False; Output Data.BitSize = 16; Output Data.DataSize = 2; Output Data.DataType = 'UINT'; Output Data.Name = 'Output Data'; Output Data.HelpString = ''; Output Data.ReadOnly = False; Output Data.BitSize = 16; Output Data.DataSize = 2; Output Data.DataType = 'UINT'; Output Data.Name = 'Output Data'; Output Data.HelpString = ''; Output Data.ReadOnly = False; Output Data.BitSize = 16; Output Data.DataSize = 2; Output Data.DataType = 'UINT'; Output Data.Name = 'Output Data'; Output Data.HelpString = ''; Output Data.ReadOnly = False; Output Data.BitSize = 16; Output Data.DataSize = 2; Output Data.DataType = 'UINT'; Output Data.Name = 'Output Data'; Output Data.HelpString = '';
              Output Data.ReadOnly = False; Output Data.BitSize = 16; Output Data.DataSize = 2; Output Data.DataType = 'UINT'; Output Data.Name = 'Output Data'; Output Data.HelpString = ''; Output Data.ReadOnly = False; Output Data.BitSize = 16; Output Data.DataSize = 2; Output Data.DataType = 'UINT'; Output Data.Name = 'Output Data'; Output Data.HelpString = ''; Output Data.ReadOnly = False; Output Data.BitSize = 16; Output Data.DataSize = 2; Output Data.DataType = 'UINT'; Output Data.Name = 'Output Data'; Output Data.HelpString = ''; Output Data.ReadOnly = False; Output Data.BitSize = 16; Output Data.DataSize = 2; Output Data.DataType = 'UINT'; Output Data.Name = 'Output Data'; Output Data.HelpString = ''; Output Data.ReadOnly = False; Output Data.BitSize = 16; Output Data.DataSize = 2; Output Data.DataType = 'UINT'; Output Data.Name = 'Output Data'; Output Data.HelpString = ''; Output Data.ReadOnly = False; Output Data.BitSize = 16; Output Data.DataSize = 2; Output Data.DataType = 'UINT'; Output Data.Name = 'Output Data'; Output Data.HelpString = ''; Output Data.ReadOnly = False; Output Data.BitSize = 16; Output Data.DataSize = 2; Output Data.DataType = 'UINT';
              Output Data.Name = 'Output Data'; Output Data.HelpString = ''; Output Data.ReadOnly = False; Output Data.BitSize = 16; Output Data.DataSize = 2; Output Data.DataType = 'UINT'; Output Data.Name = 'Output Data'; Output Data.HelpString = ''; Output Data.ReadOnly = False; Output Data.BitSize = 16; Output Data.DataSize = 2; Output Data.DataType = 'UINT'; Output Data.Name = 'Output Data'; Output Data.HelpString = ''; Output Data.ReadOnly = False; Output Data.BitSize = 16; Output Data.DataSize = 2; Output Data.DataType = 'UINT'; Output Data.Name = 'Output Data'; Output Data.HelpString = ''; Output Data.ReadOnly = False; Output Data.BitSize = 16; Output Data.DataSize = 2; Output Data.DataType = 'UINT'; Output Data.Name = 'Output Data'; Output Data.HelpString = ''; Output Data.ReadOnly = False; Output Data.BitSize = 16; Output Data.DataSize = 2; Output Data.DataType = 'UINT'; Output Data.Name = 'Output Data'; Output Data.HelpString = ''; Output Data.ReadOnly = False; Output Data.BitSize = 16; Output Data.DataSize = 2; Output Data.DataType = 'UINT'; Output Data.Name = 'Output Data'; Output Data.HelpString = ''; Output Data.ReadOnly = False; Output Data.BitSize = 16;
              Output Data.DataSize = 2; Output Data.DataType = 'UINT'; Output Data.Name = 'Output Data'; Output Data.HelpString = ''; Output Data.ReadOnly = False; Output Data.BitSize = 16; Output Data.DataSize = 2; Output Data.DataType = 'UINT'; Output Data.Name = 'Output Data'; Output Data.HelpString = ''; Output Data.ReadOnly = False; Output Data.BitSize = 16; Output Data.DataSize = 2; Output Data.DataType = 'UINT'; Output Data.Name = 'Output Data'; Output Data.HelpString = ''; Output Data.ReadOnly = False; Output Data.BitSize = 16; Output Data.DataSize = 2; Output Data.DataType = 'UINT'; Output Data.Name = 'Output Data'; Output Data.HelpString = ''; Output Data.ReadOnly = False; Output Data.BitSize = 16; Output Data.DataSize = 2; Output Data.DataType = 'UINT'; Output Data.Name = 'Output Data'; Output Data.HelpString = ''; Output Data.ReadOnly = False; Output Data.BitSize = 16; Output Data.DataSize = 2; Output Data.DataType = 'UINT'; Output Data.Name = 'Output Data'; Output Data.HelpString = ''; Output Data.ReadOnly = False; Output Data.BitSize = 16; Output Data.DataSize = 2; Output Data.DataType = 'UINT'; Output Data.Name = 'Output Data'; Output Data.HelpString = '';
              Output Data.ReadOnly = False; Output Data.BitSize = 16; Output Data.DataSize = 2; Output Data.DataType = 'UINT'; Output Data.Name = 'Output Data'; Output Data.HelpString = ''; Output Data.ReadOnly = False; Output Data.BitSize = 16; Output Data.DataSize = 2; Output Data.DataType = 'UINT'; Output Data.Name = 'Output Data'; Output Data.HelpString = ''; Output Data.ReadOnly = False; Output Data.BitSize = 16; Output Data.DataSize = 2; Output Data.DataType = 'UINT'; Output Data.Name = 'Output Data'; Output Data.HelpString = ''; Output Data.ReadOnly = False; Output Data.BitSize = 16; Output Data.DataSize = 2; Output Data.DataType = 'UINT'; Output Data.Name = 'Output Data'; Output Data.HelpString = ''; Output Data.ReadOnly = False; Output Data.BitSize = 16; Output Data.DataSize = 2; Output Data.DataType = 'UINT'; Output Data.Name = 'Output Data'; Output Data.HelpString = ''; Output Data.ReadOnly = False; Output Data.BitSize = 16; Output Data.DataSize = 2; Output Data.DataType = 'UINT'; Output Data.Name = 'Output Data'; Output Data.HelpString = ''; Output Data.ReadOnly = False; Output Data.BitSize = 16; Output Data.DataSize = 2; Output Data.DataType = 'UINT';
              Output Data.Name = 'Output Data'; Output Data.HelpString = ''; Output Data.ReadOnly = False; Output Data.BitSize = 16; Output Data.DataSize = 2; Output Data.DataType = 'UINT'; Output Data.Name = 'Output Data'; Output Data.HelpString = ''; Output Data.ReadOnly = False; Output Data.BitSize = 16; Output Data.DataSize = 2; Output Data.DataType = 'UINT'; Output Data.Name = 'Output Data'; Output Data.HelpString = ''; Output Data.ReadOnly = False; Output Data.BitSize = 16; Output Data.DataSize = 2; Output Data.DataType = 'UINT'; Output Data.Name = 'Output Data'; Output Data.HelpString = ''; Output Data.ReadOnly = False; Output Data.BitSize = 16; Output Data.DataSize = 2; Output Data.DataType = 'UINT'; Output Data.Name = 'Output Data'; Output Data.HelpString = ''; Output Data.ReadOnly = False; Output Data.BitSize = 16; Output Data.DataSize = 2; Output Data.DataType = 'UINT'; Output Data.Name = 'Output Data'; Output Data.HelpString = ''; Output Data.ReadOnly = False; Output Data.BitSize = 16; Output Data.DataSize = 2; Output Data.DataType = 'UINT'; Output Data.Name = 'Output Data'; Output Data.HelpString = ''; Output Data.ReadOnly = False; Output Data.BitSize = 16;
              Output Data.DataSize = 2; Output Data.DataType = 'UINT'; Output Data.Name = 'Output Data'; Output Data.HelpString = ''; Output Data.ReadOnly = False; Output Data.BitSize = 16; Output Data.DataSize = 2; Output Data.DataType = 'UINT'; Output Data.Name = 'Output Data'; Output Data.HelpString = ''; Output Data.ReadOnly = False; Output Data.BitSize = 16; Output Data.DataSize = 2; Output Data.DataType = 'UINT'; Output Data.Name = 'Output Data'; Output Data.HelpString = ''; Output Data.ReadOnly = False; Output Data.BitSize = 16; Output Data.DataSize = 2; Output Data.DataType = 'UINT'; Output Data.Name = 'Output Data'; Output Data.HelpString = ''; Output Data.ReadOnly = False; Output Data.BitSize = 16; Output Data.DataSize = 2; Output Data.DataType = 'UINT'; Output Data.Name = 'Output Data'; Output Data.HelpString = ''; Output Data.ReadOnly = False; Output Data.BitSize = 16; Output Data.DataSize = 2; Output Data.DataType = 'UINT'; Output Data.Name = 'Output Data'; Output Data.HelpString = ''; Output Data.ReadOnly = False; Output Data.BitSize = 16; Output Data.DataSize = 2; Output Data.DataType = 'UINT'; Output Data.Name = 'Output Data'; Output Data.HelpString = '';
              Output Data.ReadOnly = False; Output Data.BitSize = 16; Output Data.DataSize = 2; Output Data.DataType = 'UINT'; Output Data.Name = 'Output Data'; Output Data.HelpString = ''; Output Data.ReadOnly = False; Output Data.BitSize = 16; Output Data.DataSize = 2; Output Data.DataType = 'UINT'; Output Data.Name = 'Output Data'; Output Data.HelpString = ''; Output Data.ReadOnly = False; Output Data.BitSize = 16; Output Data.DataSize = 2; Output Data.DataType = 'UINT'; Output Data.Name = 'Output Data'; Output Data.HelpString = ''; Output Data.ReadOnly = False; Output Data.BitSize = 16; Output Data.DataSize = 2; Output Data.DataType = 'UINT'; Output Data.Name = 'Output Data'; Output Data.HelpString = ''; Output Data.ReadOnly = False; Output Data.BitSize = 16; Output Data.DataSize = 2; Output Data.DataType = 'UINT'; Output Data.Name = 'Output Data'; Output Data.HelpString = ''; Output Data.ReadOnly = False; Output Data.BitSize = 16; Output Data.DataSize = 2; Output Data.DataType = 'UINT'; Output Data.Name = 'Output Data'; Output Data.HelpString = ''; Output Data.ReadOnly = False; Output Data.BitSize = 16; Output Data.DataSize = 2; Output Data.DataType = 'UINT';
              Output Data.Name = 'Output Data'; Output Data.HelpString = ''; Output Data.ReadOnly = False; Output Data.BitSize = 16; Output Data.DataSize = 2; Output Data.DataType = 'UINT'; Output Data.Name = 'Output Data'; Output Data.HelpString = ''; Output Data.ReadOnly = False; Output Data.BitSize = 16; Output Data.DataSize = 2; Output Data.DataType = 'UINT'; Output Data.Name = 'Output Data'; Output Data.HelpString = ''; Output Data.ReadOnly = False; Output Data.BitSize = 16; Output Data.DataSize = 2; Output Data.DataType = 'UINT'; Output Data.Name = 'Output Data'; Output Data.HelpString = ''; Output Data.ReadOnly = False; Output Data.BitSize = 16; Output Data.DataSize = 2; Output Data.DataType = 'UINT'; Output Data.Name = 'Output Data'; Output Data.HelpString = ''; Output Data.ReadOnly = False; Output Data.BitSize = 16; Output Data.DataSize = 2; Output Data.DataType = 'UINT'; Output Data.Name = 'Output Data'; Output Data.HelpString = ''; Output Data.ReadOnly = False; Output Data.BitSize = 16; Output Data.DataSize = 2; Output Data.DataType = 'UINT'; Output Data.Name = 'Output Data'; Output Data.HelpString = ''; Output Data.ReadOnly = False; Output Data.BitSize = 16;
              Output Data.DataSize = 2; Output Data.DataType = 'UINT'; Output Data.Name = 'Output Data'; Output Data.HelpString = ''; Output Data.ReadOnly = False; Output Data.BitSize = 16; Output Data.DataSize = 2; Output Data.DataType = 'UINT'; Output Data.Name = 'Output Data'; Output Data.HelpString = ''; Output Data.ReadOnly = False; Output Data.BitSize = 16; Output Data.DataSize = 2; Output Data.DataType = 'UINT'; Output Data.Name = 'Output Data'; Output Data.HelpString = ''; Output Data.ReadOnly = False; Output Data.BitSize = 16; Output Data.DataSize = 2; Output Data.DataType = 'UINT'; Output Data.Name = 'Output Data'; Output Data.HelpString = ''; Output Data.ReadOnly = False; Output Data.BitSize = 16; Output Data.DataSize = 2; Output Data.DataType = 'UINT'; Output Data.Name = 'Output Data'; Output Data.HelpString = ''; Output Data.ReadOnly = False; Output Data.BitSize = 16; Output Data.DataSize = 2; Output Data.DataType = 'UINT'; Output Data.Name = 'Output Data'; Output Data.HelpString = ''; Output Data.ReadOnly = False; Output Data.BitSize = 16; Output Data.DataSize = 2; Output Data.DataType = 'UINT'; Output Data.Name = 'Output Data'; Output Data.HelpString = '';
              Output Data.ReadOnly = False; Output Data.BitSize = 16; Output Data.DataSize = 2; Output Data.DataType = 'UINT'; Output Data.Name = 'Output Data'; Output Data.HelpString = ''; Output Data.ReadOnly = False; Output Data.BitSize = 16; Output Data.DataSize = 2; Output Data.DataType = 'UINT'; Output Data.Name = 'Output Data'; Output Data.HelpString = ''; Output Data.ReadOnly = False; Output Data.BitSize = 16; Output Data.DataSize = 2; Output Data.DataType = 'UINT'; Output Data.Name = 'Output Data'; Output Data.HelpString = ''; Output Data.ReadOnly = False; Output Data.BitSize = 16; Output Data.DataSize = 2; Output Data.DataType = 'UINT'; Output Data.Name = 'Output Data'; Output Data.HelpString = ''; Output Data.ReadOnly = False; Output Data.BitSize = 16; Output Data.DataSize = 2; Output Data.DataType = 'UINT'; Output Data.Name = 'Output Data'; Output Data.HelpString = ''; Output Data.ReadOnly = False; Output Data.BitSize = 16; Output Data.DataSize = 2; Output Data.DataType = 'UINT'; Output Data.Name = 'Output Data'; Output Data.HelpString = ''; Output Data.ReadOnly = False; Output Data.BitSize = 16; Output Data.DataSize = 2; Output Data.DataType = 'UINT';
              Output Data.Name = 'Output Data'; Output Data.HelpString = ''; Output Data.ReadOnly = False; Output Data.BitSize = 16; Output Data.DataSize = 2; Output Data.DataType = 'UINT'; Output Data.Name = 'Output Data'; Output Data.HelpString = ''; Output Data.ReadOnly = False; Output Data.BitSize = 16; Output Data.DataSize = 2; Output Data.DataType = 'UINT'; Output Data.Name = 'Output Data'; Output Data.HelpString = ''; Output Data.ReadOnly = False; Output Data.BitSize = 16; Output Data.DataSize = 2; Output Data.DataType = 'UINT'; Output Data.Name = 'Output Data'; Output Data.HelpString = ''; Output Data.ReadOnly = False; Output Data.BitSize = 16; Output Data.DataSize = 2; Output Data.DataType = 'UINT'; Output Data.Name = 'Output Data'; Output Data.HelpString = ''; Output Data.ReadOnly = False; Output Data.BitSize = 16; Output Data.DataSize = 2; Output Data.DataType = 'UINT'; Output Data.Name = 'Output Data'; Output Data.HelpString = ''; Output Data.ReadOnly = False; Output Data.BitSize = 16; Output Data.DataSize = 2; Output Data.DataType = 'UINT'; Output Data.Name = 'Output Data'; Output Data.HelpString = ''; Output Data.ReadOnly = False; Output Data.BitSize = 16;
              Output Data.DataSize = 2; Output Data.DataType = 'UINT'; Output Data.Name = 'Output Data'; Output Data.HelpString = ''; Output Data.ReadOnly = False; Output Data.BitSize = 16; Output Data.DataSize = 2; Output Data.DataType = 'UINT'; Output Data.Name = 'Output Data'; Output Data.HelpString = ''; Output Data.ReadOnly = False; Output Data.BitSize = 16; Output Data.DataSize = 2; Output Data.DataType = 'UINT'; Output Data.Name = 'Output Data'; Output Data.HelpString = ''; Output Data.ReadOnly = False; Output Data.BitSize = 16; Output Data.DataSize = 2; Output Data.DataType = 'UINT'; Output Data.Name = 'Output Data'; Output Data.HelpString = ''; Output Data.ReadOnly = False; Output Data.BitSize = 16; Output Data.DataSize = 2; Output Data.DataType = 'UINT'; Output Data.Name = 'Output Data'; Output Data.HelpString = ''; Output Data.ReadOnly = False; Output Data.BitSize = 16; Output Data.DataSize = 2; Output Data.DataType = 'UINT'; Output Data.Name = 'Output Data'; Output Data.HelpString = ''; Output Data.ReadOnly = False; Output Data.BitSize = 16; Output Data.DataSize = 2; Output Data.DataType = 'UINT'; Output Data.Name = 'Output Data'; Output Data.HelpString = '';
              Output Data.ReadOnly = False; Output Data.BitSize = 16; Output Data.DataSize = 2; Output Data.DataType = 'UINT'; Output Data.Name = 'Output Data'; Output Data.HelpString = ''; Output Data.ReadOnly = False; Output Data.BitSize = 16; Output Data.DataSize = 2; Output Data.DataType = 'UINT'; Output Data.Name = 'Output Data'; Output Data.HelpString = ''; Output Data.ReadOnly = False; Output Data.BitSize = 16; Output Data.DataSize = 2; Output Data.DataType = 'UINT'; Output Data.Name = 'Output Data'; Output Data.HelpString = ''; Output Data.ReadOnly = False; Output Data.BitSize = 16; Output Data.DataSize = 2; Output Data.DataType = 'UINT'; Output Data.Name = 'Output Data'; Output Data.HelpString = ''; Output Data.ReadOnly = False; Output Data.BitSize = 16; Output Data.DataSize = 2; Output Data.DataType = 'UINT'; Output Data.Name = 'Output Data'; Output Data.HelpString = ''; Output Data.ReadOnly = False; Output Data.BitSize = 16; Output Data.DataSize = 2; Output Data.DataType = 'UINT'; Output Data.Name = 'Output Data'; Output Data.HelpString = ''; Output Data.ReadOnly = False; Output Data.BitSize = 16; Output Data.DataSize = 2; Output Data.DataType = 'UINT';
              Output Data.Name = 'Output Data'; Output Data.HelpString = ''; Output Data.ReadOnly = False; Output Data.BitSize = 16; Output Data.DataSize = 2; Output Data.DataType = 'UINT'; Output Data.Name = 'Output Data'; Output Data.HelpString = ''; Output Data.ReadOnly = False; Output Data.BitSize = 16; Output Data.DataSize = 2; Output Data.DataType = 'UINT'; Output Data.Name = 'Output Data'; Output Data.HelpString = ''; Output Data.ReadOnly = False; Output Data.BitSize = 16; Output Data.DataSize = 2; Output Data.DataType = 'UINT'; Output Data.Name = 'Output Data'; Output Data.HelpString = ''; Output Data.ReadOnly = False; Output Data.BitSize = 16; Output Data.DataSize = 2; Output Data.DataType = 'UINT'; Output Data.Name = 'Output Data'; Output Data.HelpString = ''; Output Data.ReadOnly = False; Output Data.BitSize = 16; Output Data.DataSize = 2; Output Data.DataType = 'UINT'; Output Data.Name = 'Output Data'; Output Data.HelpString = ''; Output Data.ReadOnly = False; Output Data.BitSize = 16; Output Data.DataSize = 2; Output Data.DataType = 'UINT'; Output Data.Name = 'Output Data'; Output Data.HelpString = ''; Output Data.ReadOnly = False; Output Data.BitSize = 16;
              Output Data.DataSize = 2; Output Data.DataType = 'UINT'; Output Data.Name = 'Output Data'; Output Data.HelpString = ''; Output Data.ReadOnly = False; Output Data.BitSize = 16; Output Data.DataSize = 2; Output Data.DataType = 'UINT'; Output Data.Name = 'Output Data'; Output Data.HelpString = ''; Output Data.ReadOnly = False; Output Data.BitSize = 16; Output Data.DataSize = 2; Output Data.DataType = 'UINT'; Output Data.Name = 'Output Data'; Output Data.HelpString = ''; Output Data.ReadOnly = False; Output Data.BitSize = 16; Output Data.DataSize = 2; Output Data.DataType = 'UINT'; Output Data.Name = 'Output Data'; Output Data.HelpString = ''; Output Data.ReadOnly = False; Output Data.BitSize = 16; Output Data.DataSize = 2; Output Data.DataType = 'UINT'; Output Data.Name = 'Output Data'; Output Data.HelpString = ''; Output Data.ReadOnly = False; Output Data.BitSize = 16; Output Data.DataSize = 2; Output Data.DataType = 'UINT'; Output Data.Name = 'Output Data'; Output Data.HelpString = ''; Output Data.ReadOnly = False; Output Data.BitSize = 16; Output Data.DataSize = 2; Output Data.DataType = 'UINT'; Output Data.Name = 'Output Data'; Output Data.HelpString = '';
              Output Data.ReadOnly = False; Output Data.BitSize = 16; Output Data.DataSize = 2; Output Data.DataType = 'UINT'; Output Data.Name = 'Output Data'; Output Data.HelpString = ''; Output Data.ReadOnly = False; Output Data.BitSize = 16; Output Data.DataSize = 2; Output Data.DataType = 'UINT'; Output Data.Name = 'Output Data'; Output Data.HelpString = ''; Output Data.ReadOnly = False; Output Data.BitSize = 16; Output Data.DataSize = 2; Output Data.DataType = 'UINT'; Output Data.Name = 'Output Data'; Output Data.HelpString = ''; Output Data.ReadOnly = False; Output Data.BitSize = 16; Output Data.DataSize = 2; Output Data.DataType = 'UINT'; Output Data.Name = 'Output Data'; Output Data.HelpString = ''; Output Data.ReadOnly = False; Output Data.BitSize = 16; Output Data.DataSize = 2; Output Data.DataType = 'UINT'; Output Data.Name = 'Output Data'; Output Data.HelpString = ''; Output Data.ReadOnly = False; Output Data.BitSize = 16; Output Data.DataSize = 2; Output Data.DataType = 'UINT'; Output Data.Name = 'Output Data'; Output Data.HelpString = ''; Output Data.ReadOnly = False; Output Data.BitSize = 16; Output Data.DataSize = 2; Output Data.DataType = 'UINT';
              Output Data.Name = 'Output Data'; Output Data.HelpString = ''; Output Data.ReadOnly = False; Output Data.BitSize = 16; Output Data.DataSize = 2; Output Data.DataType = 'UINT'; Output Data.Name = 'Output Data'; Output Data.HelpString = ''; Output Data.ReadOnly = False; Output Data.BitSize = 16; Output Data.DataSize = 2; Output Data.DataType = 'UINT'; Output Data.Name = 'Output Data'; Output Data.HelpString = ''; Output Data.ReadOnly = False; Output Data.BitSize = 16; Output Data.DataSize = 2; Output Data.DataType = 'UINT'; Output Data.Name = 'Output Data'; Output Data.HelpString = ''; Output Data.ReadOnly = False; Output Data.BitSize = 16; Output Data.DataSize = 2; Output Data.DataType = 'UINT'; Output Data.Name = 'Output Data'; Output Data.HelpString = ''; Output Data.ReadOnly = False; Output Data.BitSize = 16; Output Data.DataSize = 2; Output Data.DataType = 'UINT'; Output Data.Name = 'Output Data'; Output Data.HelpString = ''; Output Data.ReadOnly = False; Output Data.BitSize = 16; Output Data.DataSize = 2; Output Data.DataType = 'UINT'; Output Data.Name = 'Output Data'; Output Data.HelpString = ''; Output Data.ReadOnly = False; Output Data.BitSize = 16;
              Output Data.DataSize = 2; Output Data.DataType = 'UINT'; Output Data.Name = 'Output Data'; Output Data.HelpString = ''; Output Data.ReadOnly = False; Output Data.BitSize = 16; Output Data.DataSize = 2; Output Data.DataType = 'UINT'; Output Data.Name = 'Output Data'; Output Data.HelpString = ''; Output Data.ReadOnly = False; Output Data.BitSize = 16; Output Data.DataSize = 2; Output Data.DataType = 'UINT'; Output Data.Name = 'Output Data'; Output Data.HelpString = ''; Output Data.ReadOnly = False; Output Data.BitSize = 16; Output Data.DataSize = 2; Output Data.DataType = 'UINT'; ConfigVersion = 50660864
            input  Application.GL_Variables.pDB1_WORD1 : UINT  // Input Data
            input  Application.GL_Variables.pDB1_WORD2 : UINT  // Input Data
            input  Application.GL_Variables.pDB1_WORD3 : UINT  // Input Data
            input  Application.GL_Variables.tDB1_WORD1 AT %IW98 : UINT  // Input Data
            input  Application.GL_Variables.tDB1_WORD2 AT %IW99 : UINT  // Input Data
            input  Application.GL_Variables.vDB1_WORD3 : UINT  // Input Data
            input  Application.GL_Variables.vDB1_WORD2 : UINT  // Input Data
            input  Application.GL_Variables.vDB1_WORD1 : UINT  // Input Data
            input  Application.GL_Variables.pDB2_WORD1 : UINT  // Input Data
            input  Application.GL_Variables.pDB2_WORD2 : UINT  // Input Data
            input  Application.GL_Variables.pDB2_WORD3 AT %IW113 : UINT  // Input Data
            input  Application.GL_Variables.tDB2_WORD1 : UINT  // Input Data
            input  Application.GL_Variables.tDB2_WORD2 : UINT  // Input Data
            input  Application.GL_Variables.vDB2_WORD3 : UINT  // Input Data
            input  Application.GL_Variables.vDB2_WORD2 : UINT  // Input Data
            input  Application.GL_Variables.vDB2_WORD1 : UINT  // Input Data
            input  Application.GL_Variables.pDB3_WORD1 : UINT  // Input Data
            input  Application.GL_Variables.pDB3_WORD2 : UINT  // Input Data
            input  Application.GL_Variables.pDB3_WORD3 : UINT  // Input Data
            input  Application.GL_Variables.tDB3_WORD1 : UINT  // Input Data
            input  Application.GL_Variables.tDB3_WORD2 : UINT  // Input Data
            input  Application.GL_Variables.vDB3_WORD3 : UINT  // Input Data
            input  Application.GL_Variables.vDB3_WORD2 : UINT  // Input Data
            input  Application.GL_Variables.vDB3_WORD1 : UINT  // Input Data
            input  Application.GL_Variables.pDB4_WORD1 : UINT  // Input Data
            input  Application.GL_Variables.pDB4_WORD2 : UINT  // Input Data
            input  Application.GL_Variables.pDB4_WORD3 : UINT  // Input Data
            input  Application.GL_Variables.tDB4_WORD1 : UINT  // Input Data
            input  Application.GL_Variables.tDB4_WORD2 : UINT  // Input Data
            input  Application.GL_Variables.vDB4_WORD3 : UINT  // Input Data
            input  Application.GL_Variables.vDB4_WORD2 : UINT  // Input Data
            input  Application.GL_Variables.vDB4_WORD1 : UINT  // Input Data
            input  Application.GL_Variables.pDB5_WORD1 : UINT  // Input Data
            input  Application.GL_Variables.pDB5_WORD2 : UINT  // Input Data
            input  Application.GL_Variables.pDB5_WORD3 : UINT  // Input Data
            input  Application.GL_Variables.tDB5_WORD1 : UINT  // Input Data
            input  Application.GL_Variables.tDB5_WORD2 : UINT  // Input Data
            input  Application.GL_Variables.vDB5_WORD3 : UINT  // Input Data
            input  Application.GL_Variables.vDB5_WORD2 : UINT  // Input Data
            input  Application.GL_Variables.vDB5_WORD1 : UINT  // Input Data
            input  Application.GL_Variables.tSD9000_WORD1 : UINT  // Input Data
            input  Application.GL_Variables.tSD9000_WORD2 : UINT  // Input Data
            input  Application.GL_Variables.SD9000_Flow : UINT  // Input Data
            input  Application.GL_Variables.SD9000_Temp AT %IW178 : UINT  // Input Data
            input  Application.GL_Variables.pDG_WORD1 : UINT  // Input Data
            input  Application.GL_Variables.pDG_WORD2 : UINT  // Input Data
            input  Application.GL_Variables.pDG_WORD3 : UINT  // Input Data
            input  Application.GL_Variables.tDG_WORD1 : UINT  // Input Data
            input  Application.GL_Variables.tDG_WORD2 : UINT  // Input Data
            input  Application.GL_Variables.vDG_WORD3 : UINT  // Input Data
            input  Application.GL_Variables.vDG_WORD2 : UINT  // Input Data
            input  Application.GL_Variables.vDG_WORD1 : UINT  // Input Data
            unmapped channels: Input Data, Input Data, Input Data, Input Data, Input Data, Input Data, Input Data, Input Data, Input Data, Input Data, Input Data, Input Data, Input Data, Input Data, Input Data, Input Data, Input Data, Input Data, Input Data, Input Data, Input Data, Input Data, Input Data, Input Data, Input Data, Input Data, Input Data, Input Data, Input Data, Input Data, Input Data, Input Data, Input Data, Input Data, Input Data, Input Data, Input Data, Input Data, Input Data, Input Data,
              Input Data, Input Data, Input Data, Input Data, Input Data, Input Data, Input Data, Input Data, Input Data, Input Data, Input Data, Input Data, Input Data, Input Data, Input Data, Input Data, Input Data, Input Data, Input Data, Input Data, Input Data, Input Data, Input Data, Input Data, Input Data, Input Data, Input Data, Input Data, Input Data, Input Data, Input Data, Input Data, Input Data, Input Data, Input Data, Input Data, Input Data, Input Data, Input Data, Input Data,
              Input Data, Input Data, Input Data, Input Data, Input Data, Input Data, Input Data, Input Data, Input Data, Input Data, Input Data, Input Data, Input Data, Input Data, Input Data, Input Data, Input Data, Input Data, Input Data, Input Data, Input Data, Input Data, Input Data, Input Data, Input Data, Input Data, Input Data, Input Data, Input Data, Input Data, Input Data, Input Data, Input Data, Input Data, Input Data, Input Data, Input Data, Input Data, Input Data, Input Data,
              Input Data, Input Data, Input Data, Input Data, Input Data, Input Data, Input Data, Input Data, Input Data, Input Data, Input Data, Input Data, Input Data, Input Data, Input Data, Input Data, Input Data, Input Data, Input Data, Input Data, Input Data, Input Data, Input Data, Input Data, Input Data, Input Data, Input Data, Input Data, Input Data, Input Data, Input Data, Input Data, Input Data, Input Data, Input Data, Input Data, Input Data, Input Data, Input Data, Input Data,
              Input Data, Input Data, Input Data, Input Data, Input Data, Input Data, Input Data, Input Data, Input Data, Input Data, Input Data, Output Data, Output Data, Output Data, Output Data, Output Data, Output Data, Output Data, Output Data, Output Data, Output Data, Output Data, Output Data, Output Data, Output Data, Output Data, Output Data, Output Data, Output Data, Output Data, Output Data, Output Data, Output Data, Output Data, Output Data, Output Data, Output Data, Output Data, Output Data, Output Data,
              Output Data, Output Data, Output Data, Output Data, Output Data, Output Data, Output Data, Output Data, Output Data, Output Data, Output Data, Output Data, Output Data, Output Data, Output Data, Output Data, Output Data, Output Data, Output Data, Output Data, Output Data, Output Data, Output Data, Output Data, Output Data, Output Data, Output Data, Output Data, Output Data, Output Data, Output Data, Output Data, Output Data, Output Data, Output Data, Output Data, Output Data, Output Data, Output Data, Output Data,
              Output Data, Output Data, Output Data, Output Data, Output Data, Output Data, Output Data, Output Data, Output Data, Output Data, Output Data, Output Data, Output Data, Output Data, Output Data, Output Data, Output Data, Output Data, Output Data, Output Data, Output Data, Output Data, Output Data, Output Data, Output Data, Output Data, Output Data, Output Data, Output Data, Output Data, Output Data, Output Data, Output Data, Output Data, Output Data, Output Data, Output Data, Output Data, Output Data, Output Data,
              Output Data, Output Data, Output Data, Output Data, Output Data, Output Data, Output Data, Output Data, Output Data, Output Data, Output Data, Output Data, Output Data, Output Data, Output Data, Output Data, Output Data, Output Data, Output Data, Output Data, Output Data, Output Data, Output Data, Output Data, Output Data, Output Data, Output Data, Output Data, Output Data, Output Data, Output Data, Output Data, Output Data, Output Data, Output Data, Output Data, Output Data, Output Data, Output Data, Output Data,
              Output Data, Output Data
    SPI
    SoftMotion General Axis Pool
    I²C
    GPIOs_A_B : GPIOs A/B, CODESYS, version 4.21.0.0
        unmapped channels: digital inputs (GPIO0..GPIO31), digital outputs (GPIO0..GPIO31)
    Camera device
      <Empty>
  text list GlobalTextList
*)

// Device/Application/GL_Variables
{attribute 'qualified_only'}
VAR_GLOBAL

// DB1 ::::::::::::::::::::::::::::::::::::::::::::::::::::::::::::
	// Voltage Preocess DataBytes
		vDB1_WORD1						: ARRAY[0..1] OF BYTE;
		vDB1_WORD2						: ARRAY[0..1] OF BYTE;
		vDB1_WORD3						: ARRAY[0..1] OF BYTE;
		vDB1_Voltage_PD					: ARRAY[0..3] OF BYTE;
		vDB1_Voltage					: DWORD;
		vDB1_Voltage_Value				: REAL;
	
	// Temperature process DataBytes
		tDB1_WORD1						: ARRAY[0..1] OF BYTE;
		tDB1_WORD2						: ARRAY[0..1] OF BYTE;
		tDB1_Temp						: DWORD;
		tDB1_Temp_Value					: REAL;	

	// Pressure Process DataBytes
		pDB1_WORD1						: ARRAY[0..1] OF BYTE;
		pDB1_WORD2						: ARRAY[0..1] OF BYTE;
		pDB1_WORD3						: ARRAY[0..1] OF BYTE;
		pDB1_Pressure_PD				: ARRAY[0..3] OF BYTE;	
		pDB1_Pressure					: DWORD;
		pDB1_Pressure_Value				: REAL;
	
// DB2 ::::::::::::::::::::::::::::::::::::::::::::::::::::::::::::

	// Voltage Preocess DataBytes
		vDB2_WORD1						: ARRAY[0..1] OF BYTE;
		vDB2_WORD2						: ARRAY[0..1] OF BYTE;
		vDB2_WORD3						: ARRAY[0..1] OF BYTE;
		vDB2_Voltage_PD					: ARRAY[0..3] OF BYTE;
		vDB2_Voltage					: DWORD;
		vDB2_Voltage_Value				: REAL;
	
	// Temperature process DataBytes
		tDB2_WORD1						: ARRAY[0..1] OF BYTE;
		tDB2_WORD2						: ARRAY[0..1] OF BYTE;
		tDB2_Temp						: DWORD;
		tDB2_Temp_Value					: REAL;	

	// Pressure Process DataBytes
		pDB2_WORD1						: ARRAY[0..1] OF BYTE;
		pDB2_WORD2						: ARRAY[0..1] OF BYTE;
		pDB2_WORD3						: ARRAY[0..1] OF BYTE;
		pDB2_Pressure_PD				: ARRAY[0..3] OF BYTE;	
		pDB2_Pressure					: DWORD;
		pDB2_Pressure_Value				: REAL;
	
// DB3 ::::::::::::::::::::::::::::::::::::::::::::::::::::::::::::::::
	// Voltage Preocess DataBytes
		vDB3_WORD1						: ARRAY[0..1] OF BYTE;
		vDB3_WORD2						: ARRAY[0..1] OF BYTE;
		vDB3_WORD3						: ARRAY[0..1] OF BYTE;
		vDB3_Voltage_PD					: ARRAY[0..3] OF BYTE;
		vDB3_Voltage					: DWORD;
		vDB3_Voltage_Value				: REAL;
	
	// Temperature process DataBytes
		tDB3_WORD1						: ARRAY[0..1] OF BYTE;
		tDB3_WORD2						: ARRAY[0..1] OF BYTE;
		tDB3_Temp						: DWORD;
		tDB3_Temp_Value					: REAL;	

	// Pressure Process DataBytes
		pDB3_WORD1						: ARRAY[0..1] OF BYTE;
		pDB3_WORD2						: ARRAY[0..1] OF BYTE;
		pDB3_WORD3						: ARRAY[0..1] OF BYTE;
		pDB3_Pressure_PD				: ARRAY[0..3] OF BYTE;	
		pDB3_Pressure					: DWORD;
		pDB3_Pressure_Value				: REAL;
		
// DB4 ::::::::::::::::::::::::::::::::::::::::::::::::::::::::::::::::::::::::		
	
	// Voltage Process DataBytes
		vDB4_WORD1						: ARRAY[0..1] OF BYTE;
		vDB4_WORD2						: ARRAY[0..1] OF BYTE;
		vDB4_WORD3						: ARRAY[0..1] OF BYTE;
		vDB4_Voltage_PD					: ARRAY[0..3] OF BYTE;
		vDB4_Voltage					: DWORD;
		vDB4_Voltage_Value				: REAL;
	
	// Temperature Process DataBytes
		tDB4_WORD1						: ARRAY[0..1] OF BYTE;
		tDB4_WORD2						: ARRAY[0..1] OF BYTE;
		tDB4_Temp						: DWORD;
		tDB4_Temp_Value					: REAL;	

	// Pressure Process DataBytes
		pDB4_WORD1						: ARRAY[0..1] OF BYTE;
		pDB4_WORD2						: ARRAY[0..1] OF BYTE;
		pDB4_WORD3						: ARRAY[0..1] OF BYTE;
		pDB4_Pressure_PD				: ARRAY[0..3] OF BYTE;	
		pDB4_Pressure					: DWORD;
		pDB4_Pressure_Value				: REAL;
		
// DB5 :::::::::::::::::::::::::::::::::::::::::::::::::::::::::::::::::::::::::::::::
	
	// Voltage Preocess DataBytes
		vDB5_WORD1						: ARRAY[0..1] OF BYTE;
		vDB5_WORD2						: ARRAY[0..1] OF BYTE;
		vDB5_WORD3						: ARRAY[0..1] OF BYTE;
		vDB5_Voltage_PD					: ARRAY[0..3] OF BYTE;
		vDB5_Voltage					: DWORD;
		vDB5_Voltage_Value				: REAL;
	
	// Temperature process DataBytes
		tDB5_WORD1						: ARRAY[0..1] OF BYTE;
		tDB5_WORD2						: ARRAY[0..1] OF BYTE;
		tDB5_Temp						: DWORD;
		tDB5_Temp_Value					: REAL;	

	// Pressure Process DataBytes
		pDB5_WORD1						: ARRAY[0..1] OF BYTE;
		pDB5_WORD2						: ARRAY[0..1] OF BYTE;
		pDB5_WORD3						: ARRAY[0..1] OF BYTE;
		pDB5_Pressure_PD				: ARRAY[0..3] OF BYTE;	
		pDB5_Pressure					: DWORD;
		pDB5_Pressure_Value				: REAL;
		
// Totalizer Process DataBytes
	tSD9000_WORD1					: WORD;
	tSD9000_WORD2					: WORD;
	tSD9000_Tot						: DWORD;
	tSD9000_Totalizer_Value			: REAL;
	
	SD9000_Flow						: UINT;
	SD9000_Flow_value				: REAL;
	
	SD9000_Temp						: UINT;
	SD9000_Temp_Value				: REAL;
	
// Main Supply DG :::::::::::::::::::::::::::::::::::::::::::::::::::::::::::::::::::::::::::::::
	
	// Voltage Preocess DataBytes
		vDG_WORD1						: ARRAY[0..1] OF BYTE;
		vDG_WORD2						: ARRAY[0..1] OF BYTE;
		vDG_WORD3						: ARRAY[0..1] OF BYTE;
		vDG_Voltage_PD					: ARRAY[0..3] OF BYTE;
		vDG_Voltage						: DWORD;
		vDG_Voltage_Value				: REAL;
	
	// Temperature process DataBytes
		tDG_WORD1						: ARRAY[0..1] OF BYTE;
		tDG_WORD2						: ARRAY[0..1] OF BYTE;
		tDG_Temp						: DWORD;
		tDG_Temp_Value					: REAL;	

	// Pressure Process DataBytes
		pDG_WORD1						: ARRAY[0..1] OF BYTE;
		pDG_WORD2						: ARRAY[0..1] OF BYTE;
		pDG_WORD3						: ARRAY[0..1] OF BYTE;
		pDG_Pressure_PD					: ARRAY[0..3] OF BYTE;	
		pDG_Pressure					: DWORD;
		pDG_Pressure_Value				: REAL;
		
END_VAR

// Device/Application/Main
PROGRAM Main
VAR
	i,j,a,b,c,d,e,f,g,h,k,l				: INT;
	len									: INT := 4;
	PackData							: IOLink_Dashboard;
	DisplayData							: IOLink_Dashboard;
		
END_VAR


// Display Data is received as a 16 Bytes DWORD as [01BC 15FD AB01 41E0 5D65 0141 BF02 5900]
	
	
//DB1 :::::::::::::::::::::::::::::::::::::::::::::::::::::::::::::::::::::::::::::::::::::::
	// DB1 Voltage data (IN HEX VALUE)
		FOR i := 0 TO len DO	
			GL_Variables.vDB1_Voltage_PD[3] := GL_Variables.vDB1_WORD1[1];	//41 
			GL_Variables.vDB1_Voltage_PD[2] := GL_Variables.vDB1_WORD2[0];	//BF
			GL_Variables.vDB1_Voltage_PD[1] := GL_Variables.vDB1_WORD2[1];	//02
			GL_Variables.vDB1_Voltage_PD[0] := GL_Variables.vDB1_WORD3[0];	//59
		END_FOR
		
	// DB1 Pressure data
		FOR j := 0 TO len DO	
			GL_Variables.pDB1_Pressure_PD[3] := GL_Variables.pDB1_WORD1[0];	//BC
			GL_Variables.pDB1_Pressure_PD[2] := GL_Variables.pDB1_WORD2[0];	//15
			GL_Variables.pDB1_Pressure_PD[1] := GL_Variables.pDB1_WORD2[1];	//FD
			GL_Variables.pDB1_Pressure_PD[0] := GL_Variables.pDB1_WORD3[1];	//AB
		END_FOR
//DB2 ::::::::::::::::::::::::::::::::::::::::::::::::::::::::::::::::::::::::::::::::::::::::::

	// Voltage data 
		FOR a := 0 TO len DO	
			GL_Variables.vDB2_Voltage_PD[3] := GL_Variables.vDB2_WORD1[1];	
			GL_Variables.vDB2_Voltage_PD[2] := GL_Variables.vDB2_WORD2[0];	
			GL_Variables.vDB2_Voltage_PD[1] := GL_Variables.vDB2_WORD2[1];	
			GL_Variables.vDB2_Voltage_PD[0] := GL_Variables.vDB2_WORD3[0];	
		END_FOR
		
	// Pressure data
		FOR b := 0 TO len DO	
			GL_Variables.pDB2_Pressure_PD[3] := GL_Variables.pDB2_WORD1[0];	
			GL_Variables.pDB2_Pressure_PD[2] := GL_Variables.pDB2_WORD2[0];	
			GL_Variables.pDB2_Pressure_PD[1] := GL_Variables.pDB2_WORD2[1];	
			GL_Variables.pDB2_Pressure_PD[0] := GL_Variables.pDB2_WORD3[1];	
		END_FOR

// DB3 ::::::::::::::::::::::::::::::::::::::::::::::::::::::::::::::::::::::::::::::::::::::::
	//  Voltage data
		FOR c := 0 TO len DO	
			GL_Variables.vDB3_Voltage_PD[3] := GL_Variables.vDB3_WORD1[1];	
			GL_Variables.vDB3_Voltage_PD[2] := GL_Variables.vDB3_WORD2[0];	
			GL_Variables.vDB3_Voltage_PD[1] := GL_Variables.vDB3_WORD2[1];	
			GL_Variables.vDB3_Voltage_PD[0] := GL_Variables.vDB3_WORD3[0];	
		END_FOR
		
	// Pressure data
		FOR d := 0 TO len DO	
			GL_Variables.pDB3_Pressure_PD[3] := GL_Variables.pDB3_WORD1[0];	
			GL_Variables.pDB3_Pressure_PD[2] := GL_Variables.pDB3_WORD2[0];	
			GL_Variables.pDB3_Pressure_PD[1] := GL_Variables.pDB3_WORD2[1];	
			GL_Variables.pDB3_Pressure_PD[0] := GL_Variables.pDB3_WORD3[1];	
		END_FOR
		
//DB4 ::::::::::::::::::::::::::::::::::::::::::::::::::::::::::::::::::::::::::::::::::::::::::

	// Voltage data 
		FOR e := 0 TO len DO	
			GL_Variables.vDB4_Voltage_PD[3] := GL_Variables.vDB4_WORD1[1];	
			GL_Variables.vDB4_Voltage_PD[2] := GL_Variables.vDB4_WORD2[0];	
			GL_Variables.vDB4_Voltage_PD[1] := GL_Variables.vDB4_WORD2[1];	
			GL_Variables.vDB4_Voltage_PD[0] := GL_Variables.vDB4_WORD3[0];	
		END_FOR
		
	// Pressure data
		FOR f := 0 TO len DO	
			GL_Variables.pDB4_Pressure_PD[3] := GL_Variables.pDB4_WORD1[0];	
			GL_Variables.pDB4_Pressure_PD[2] := GL_Variables.pDB4_WORD2[0];	
			GL_Variables.pDB4_Pressure_PD[1] := GL_Variables.pDB4_WORD2[1];	
			GL_Variables.pDB4_Pressure_PD[0] := GL_Variables.pDB4_WORD3[1];	
		END_FOR
		
//DB5 ::::::::::::::::::::::::::::::::::::::::::::::::::::::::::::::::::::::::::::::::::::::::::

	// Voltage data 
		FOR g := 0 TO len DO	
			GL_Variables.vDB5_Voltage_PD[3] := GL_Variables.vDB5_WORD1[1];	
			GL_Variables.vDB5_Voltage_PD[2] := GL_Variables.vDB5_WORD2[0];	
			GL_Variables.vDB5_Voltage_PD[1] := GL_Variables.vDB5_WORD2[1];	
			GL_Variables.vDB5_Voltage_PD[0] := GL_Variables.vDB5_WORD3[0];	
		END_FOR
		
	// Pressure data
		FOR h := 0 TO len DO	
			GL_Variables.pDB5_Pressure_PD[3] := GL_Variables.pDB5_WORD1[0];	
			GL_Variables.pDB5_Pressure_PD[2] := GL_Variables.pDB5_WORD2[0];	
			GL_Variables.pDB5_Pressure_PD[1] := GL_Variables.pDB5_WORD2[1];	
			GL_Variables.pDB5_Pressure_PD[0] := GL_Variables.pDB5_WORD3[1];	
		END_FOR
		
//Main Supply DG ::::::::::::::::::::::::::::::::::::::::::::::::::::::::::::::::::::::::::::::::::::::::::

	// Voltage data 
		FOR k := 0 TO len DO	
			GL_Variables.vDG_Voltage_PD[3] := GL_Variables.vDG_WORD1[1];	
			GL_Variables.vDG_Voltage_PD[2] := GL_Variables.vDG_WORD2[0];	
			GL_Variables.vDG_Voltage_PD[1] := GL_Variables.vDG_WORD2[1];	
			GL_Variables.vDG_Voltage_PD[0] := GL_Variables.vDG_WORD3[0];	
		END_FOR
		
	// Pressure data
		FOR l := 0 TO len DO	
			GL_Variables.pDG_Pressure_PD[3] := GL_Variables.pDG_WORD1[0];	
			GL_Variables.pDG_Pressure_PD[2] := GL_Variables.pDG_WORD2[0];	
			GL_Variables.pDG_Pressure_PD[1] := GL_Variables.pDG_WORD2[1];	
			GL_Variables.pDG_Pressure_PD[0] := GL_Variables.pDG_WORD3[1];	
		END_FOR		
		
		
		
		
		
		packData.Process_Data();				//Calling ProcessData Method
		DisplayData.Dashboard_Data();			//Calling DashboardData Method

END_PROGRAM

// Device/Application/IOLink_Dashboard
FUNCTION_BLOCK IOLink_Dashboard
VAR_INPUT
END_VAR
VAR_OUTPUT
END_VAR
VAR
END_VAR

// NETWORK 1

METHOD Process_Data
VAR
	
END_VAR  // Process data is manipulated and packed to DWORD
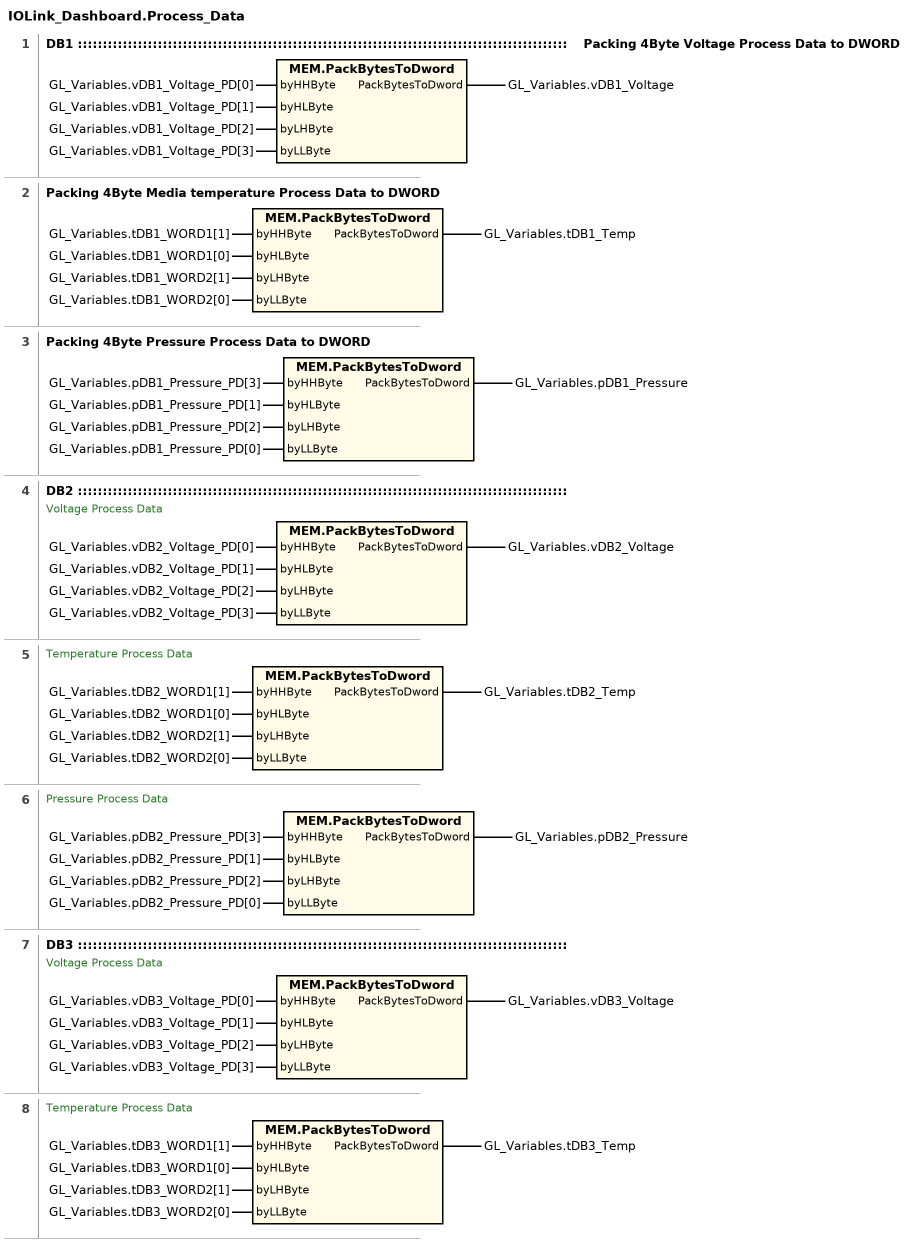
// NETWORK 1: DB1 :::::::::::::::::::::::::::::::::::::::::::::::::::::::::::::::::::::::::::::::::::::::::::::::::: Packing 4Byte Voltage Process Data to DWORD
GL_Variables.vDB1_Voltage := MEM.PackBytesToDword(byHHByte := GL_Variables.vDB1_Voltage_PD[0], byHLByte := GL_Variables.vDB1_Voltage_PD[1], byLHByte := GL_Variables.vDB1_Voltage_PD[2], byLLByte := GL_Variables.vDB1_Voltage_PD[3]);

// NETWORK 2: Packing 4Byte Media temperature Process Data to DWORD
GL_Variables.tDB1_Temp := MEM.PackBytesToDword(byHHByte := GL_Variables.tDB1_WORD1[1], byHLByte := GL_Variables.tDB1_WORD1[0], byLHByte := GL_Variables.tDB1_WORD2[1], byLLByte := GL_Variables.tDB1_WORD2[0]);

// NETWORK 3: Packing 4Byte Pressure Process Data to DWORD
GL_Variables.pDB1_Pressure := MEM.PackBytesToDword(byHHByte := GL_Variables.pDB1_Pressure_PD[3], byHLByte := GL_Variables.pDB1_Pressure_PD[1], byLHByte := GL_Variables.pDB1_Pressure_PD[2], byLLByte := GL_Variables.pDB1_Pressure_PD[0]);

// NETWORK 4: DB2 ::::::::::::::::::::::::::::::::::::::::::::::::::::::::::::::::::::::::::::::::::::::::::::::::::
// Voltage Process Data
GL_Variables.vDB2_Voltage := MEM.PackBytesToDword(byHHByte := GL_Variables.vDB2_Voltage_PD[0], byHLByte := GL_Variables.vDB2_Voltage_PD[1], byLHByte := GL_Variables.vDB2_Voltage_PD[2], byLLByte := GL_Variables.vDB2_Voltage_PD[3]);

// NETWORK 5
// Temperature Process Data
GL_Variables.tDB2_Temp := MEM.PackBytesToDword(byHHByte := GL_Variables.tDB2_WORD1[1], byHLByte := GL_Variables.tDB2_WORD1[0], byLHByte := GL_Variables.tDB2_WORD2[1], byLLByte := GL_Variables.tDB2_WORD2[0]);

// NETWORK 6
// Pressure Process Data
GL_Variables.pDB2_Pressure := MEM.PackBytesToDword(byHHByte := GL_Variables.pDB2_Pressure_PD[3], byHLByte := GL_Variables.pDB2_Pressure_PD[1], byLHByte := GL_Variables.pDB2_Pressure_PD[2], byLLByte := GL_Variables.pDB2_Pressure_PD[0]);

// NETWORK 7: DB3 ::::::::::::::::::::::::::::::::::::::::::::::::::::::::::::::::::::::::::::::::::::::::::::::::::
// Voltage Process Data
GL_Variables.vDB3_Voltage := MEM.PackBytesToDword(byHHByte := GL_Variables.vDB3_Voltage_PD[0], byHLByte := GL_Variables.vDB3_Voltage_PD[1], byLHByte := GL_Variables.vDB3_Voltage_PD[2], byLLByte := GL_Variables.vDB3_Voltage_PD[3]);

// NETWORK 8
// Temperature Process Data
GL_Variables.tDB3_Temp := MEM.PackBytesToDword(byHHByte := GL_Variables.tDB3_WORD1[1], byHLByte := GL_Variables.tDB3_WORD1[0], byLHByte := GL_Variables.tDB3_WORD2[1], byLLByte := GL_Variables.tDB3_WORD2[0]);

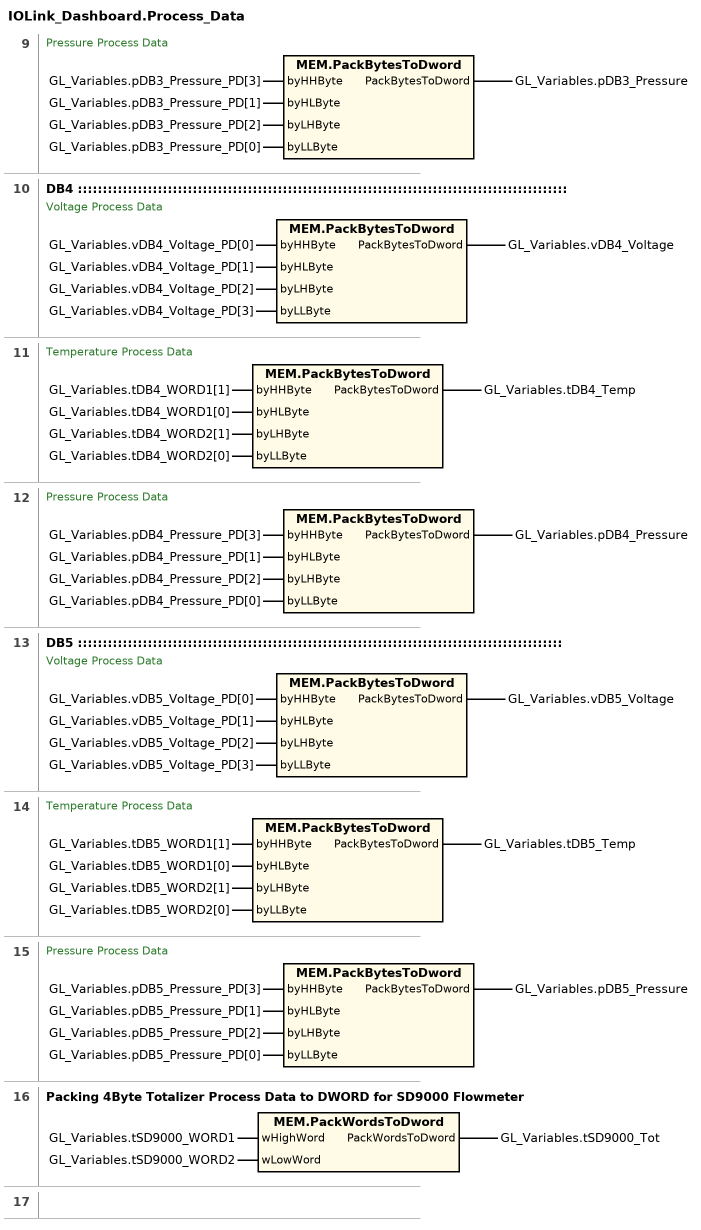
// NETWORK 9
// Pressure Process Data
GL_Variables.pDB3_Pressure := MEM.PackBytesToDword(byHHByte := GL_Variables.pDB3_Pressure_PD[3], byHLByte := GL_Variables.pDB3_Pressure_PD[1], byLHByte := GL_Variables.pDB3_Pressure_PD[2], byLLByte := GL_Variables.pDB3_Pressure_PD[0]);

// NETWORK 10: DB4 ::::::::::::::::::::::::::::::::::::::::::::::::::::::::::::::::::::::::::::::::::::::::::::::::::
// Voltage Process Data
GL_Variables.vDB4_Voltage := MEM.PackBytesToDword(byHHByte := GL_Variables.vDB4_Voltage_PD[0], byHLByte := GL_Variables.vDB4_Voltage_PD[1], byLHByte := GL_Variables.vDB4_Voltage_PD[2], byLLByte := GL_Variables.vDB4_Voltage_PD[3]);

// NETWORK 11
// Temperature Process Data
GL_Variables.tDB4_Temp := MEM.PackBytesToDword(byHHByte := GL_Variables.tDB4_WORD1[1], byHLByte := GL_Variables.tDB4_WORD1[0], byLHByte := GL_Variables.tDB4_WORD2[1], byLLByte := GL_Variables.tDB4_WORD2[0]);

// NETWORK 12
// Pressure Process Data
GL_Variables.pDB4_Pressure := MEM.PackBytesToDword(byHHByte := GL_Variables.pDB4_Pressure_PD[3], byHLByte := GL_Variables.pDB4_Pressure_PD[1], byLHByte := GL_Variables.pDB4_Pressure_PD[2], byLLByte := GL_Variables.pDB4_Pressure_PD[0]);

// NETWORK 13: DB5 :::::::::::::::::::::::::::::::::::::::::::::::::::::::::::::::::::::::::::::::::::::::::::::::::
// Voltage Process Data
GL_Variables.vDB5_Voltage := MEM.PackBytesToDword(byHHByte := GL_Variables.vDB5_Voltage_PD[0], byHLByte := GL_Variables.vDB5_Voltage_PD[1], byLHByte := GL_Variables.vDB5_Voltage_PD[2], byLLByte := GL_Variables.vDB5_Voltage_PD[3]);

// NETWORK 14
// Temperature Process Data
GL_Variables.tDB5_Temp := MEM.PackBytesToDword(byHHByte := GL_Variables.tDB5_WORD1[1], byHLByte := GL_Variables.tDB5_WORD1[0], byLHByte := GL_Variables.tDB5_WORD2[1], byLLByte := GL_Variables.tDB5_WORD2[0]);

// NETWORK 15
// Pressure Process Data
GL_Variables.pDB5_Pressure := MEM.PackBytesToDword(byHHByte := GL_Variables.pDB5_Pressure_PD[3], byHLByte := GL_Variables.pDB5_Pressure_PD[1], byLHByte := GL_Variables.pDB5_Pressure_PD[2], byLLByte := GL_Variables.pDB5_Pressure_PD[0]);

// NETWORK 16: Packing 4Byte Totalizer Process Data to DWORD for SD9000 Flowmeter
GL_Variables.tSD9000_Tot := MEM.PackWordsToDword(wHighWord := GL_Variables.tSD9000_WORD1, wLowWord := GL_Variables.tSD9000_WORD2);

// NETWORK 17

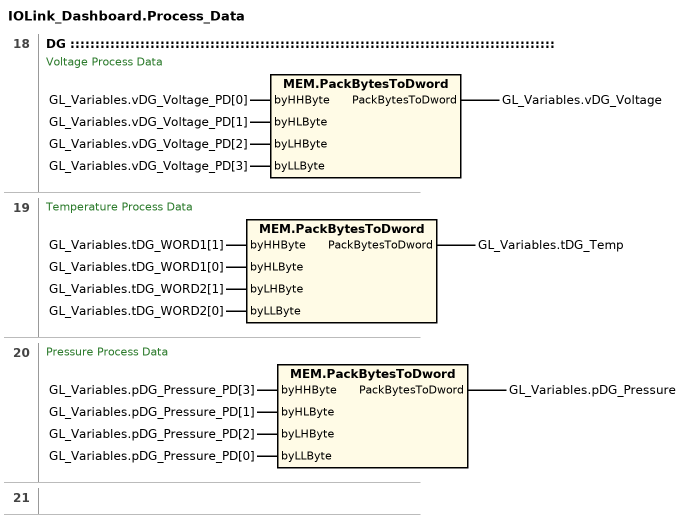
// NETWORK 18: DG :::::::::::::::::::::::::::::::::::::::::::::::::::::::::::::::::::::::::::::::::::::::::::::::::
// Voltage Process Data
GL_Variables.vDG_Voltage := MEM.PackBytesToDword(byHHByte := GL_Variables.vDG_Voltage_PD[0], byHLByte := GL_Variables.vDG_Voltage_PD[1], byLHByte := GL_Variables.vDG_Voltage_PD[2], byLLByte := GL_Variables.vDG_Voltage_PD[3]);

// NETWORK 19
// Temperature Process Data
GL_Variables.tDG_Temp := MEM.PackBytesToDword(byHHByte := GL_Variables.tDG_WORD1[1], byHLByte := GL_Variables.tDG_WORD1[0], byLHByte := GL_Variables.tDG_WORD2[1], byLLByte := GL_Variables.tDG_WORD2[0]);

// NETWORK 20
// Pressure Process Data
GL_Variables.pDG_Pressure := MEM.PackBytesToDword(byHHByte := GL_Variables.pDG_Pressure_PD[3], byHLByte := GL_Variables.pDG_Pressure_PD[1], byLHByte := GL_Variables.pDG_Pressure_PD[2], byLLByte := GL_Variables.pDG_Pressure_PD[0]);

// NETWORK 21
END_METHOD

METHOD Dashboard_Data
VAR
	DB1_vPointer				: POINTER TO REAL;		// DB1 Voltage Pointer
	DB1_tPointer				: POINTER TO REAL;		// DB1 Temperature Pointer
	DB1_pPointer				: POINTER TO REAL;		// DB1 Pressure Pointer
	
	DB2_vPointer				: POINTER TO REAL;		// DB2 Voltage Pointer
	DB2_tPointer				: POINTER TO REAL;		// DB2 Temperature Pointer
	DB2_pPointer				: POINTER TO REAL;		// DB2 Pressure Pointer
	
	DB3_vPointer				: POINTER TO REAL;		// DB3 Voltage Pointer
	DB3_tPointer				: POINTER TO REAL;		// DB3 Temperature Pointer
	DB3_pPointer				: POINTER TO REAL;		// DB3 Pressure Pointer
	
	DB4_vPointer				: POINTER TO REAL;		// DB4 Voltage Pointer
	DB4_tPointer				: POINTER TO REAL;		// DB4 Temperature Pointer
	DB4_pPointer				: POINTER TO REAL;		// DB4 Pressure Pointer
	
	DB5_vPointer				: POINTER TO REAL;		// DB5 Voltage Pointer
	DB5_tPointer				: POINTER TO REAL;		// DB5 Temperature Pointer
	DB5_pPointer				: POINTER TO REAL;		// DB5 Pressure Pointer
	
	DG_vPointer					: POINTER TO REAL;		// DG Voltage Pointer
	DG_tPointer					: POINTER TO REAL;		// DG Temperature Pointer
	DG_pPointer					: POINTER TO REAL;		// DG Pressure Pointer
	
	Totalizer					: POINTER TO REAL;		// Flowmeter Totalizer Pointer
END_VAR
// DB1 ::::::::::::::::::::::::::::::::::::::::::::::::::::::::::::::::::::::::::::::

	//1. Convert Device Supply Voltage process data to a decimal value such as 24VDC

		DB1_vPointer						:= ADR(GL_Variables.vDB1_Voltage);
		GL_Variables.vDB1_Voltage_Value		:= DB1_vPointer^;

	//2. Convert DB1 Media temperature process data to a decimal value such as 24.3°C
		DB1_tPointer						:= ADR(GL_Variables.tDB1_Temp);
		GL_Variables.tDB1_Temp_Value		:= DB1_tPointer^;

	//3. Convert DB1 Pressure process data to a decimal value such as 3.5 Bar
		DB1_pPointer							:= ADR(GL_Variables.pDB1_Pressure);
		GL_Variables.pDB1_Pressure_Value	:= DB1_pPointer^;

//DB2 :::::::::::::::::::::::::::::::::::::::::::::::::::::::::::::::::::::::::::::::::

		DB2_vPointer							:= ADR(GL_Variables.vDB2_Voltage);
		GL_Variables.vDB2_Voltage_Value			:= DB2_vPointer^;
		
		DB2_tPointer							:= ADR(GL_Variables.tDB2_Temp);
		GL_Variables.tDB2_Temp_Value			:= DB2_tPointer^;
		
		DB2_pPointer							:= ADR(GL_Variables.pDB2_Pressure);
		GL_Variables.pDB2_Pressure_Value		:= DB2_pPointer^;
// DB3 ::::::::::::::::::::::::::::::::::::::::::::::::::::::::::::::::::::::::::::::::::
		DB3_vPointer							:= ADR(GL_Variables.vDB3_Voltage);
		GL_Variables.vDB3_Voltage_Value			:= DB3_vPointer^;
		
		DB3_tPointer							:= ADR(GL_Variables.tDB3_Temp);
		GL_Variables.tDB3_Temp_Value			:= DB3_tPointer^;
		
		DB3_pPointer							:= ADR(GL_Variables.pDB3_Pressure);
		GL_Variables.pDB3_Pressure_Value		:= DB3_pPointer^;
		
//DB4 :::::::::::::::::::::::::::::::::::::::::::::::::::::::::::::::::::::::::::::::::

		DB4_vPointer							:= ADR(GL_Variables.vDB4_Voltage);
		GL_Variables.vDB4_Voltage_Value			:= DB4_vPointer^;
		
		DB4_tPointer							:= ADR(GL_Variables.tDB4_Temp);
		GL_Variables.tDB4_Temp_Value			:= DB4_tPointer^;
		
		DB4_pPointer							:= ADR(GL_Variables.pDB4_Pressure);
		GL_Variables.pDB4_Pressure_Value		:= DB4_pPointer^;
		
//DB5 :::::::::::::::::::::::::::::::::::::::::::::::::::::::::::::::::::::::::::::::::

		DB5_vPointer							:= ADR(GL_Variables.vDB5_Voltage);
		GL_Variables.vDB5_Voltage_Value			:= DB5_vPointer^;
		
		DB5_tPointer							:= ADR(GL_Variables.tDB5_Temp);
		GL_Variables.tDB5_Temp_Value			:= DB5_tPointer^;
		
		DB5_pPointer							:= ADR(GL_Variables.pDB5_Pressure);
		GL_Variables.pDB5_Pressure_Value		:= DB5_pPointer^;		

//DG :::::::::::::::::::::::::::::::::::::::::::::::::::::::::::::::::::::::::::::::::

		DG_vPointer								:= ADR(GL_Variables.vDG_Voltage);
		GL_Variables.vDG_Voltage_Value			:= DG_vPointer^;
		
		DG_tPointer								:= ADR(GL_Variables.tDG_Temp);
		GL_Variables.tDG_Temp_Value				:= DG_tPointer^;
		
		DG_pPointer								:= ADR(GL_Variables.pDG_Pressure);
		GL_Variables.pDG_Pressure_Value			:= DG_pPointer^;		
	
// Convertin SD9000 Flowmeter data to value
	Totalizer									:= ADR(GL_VAriables.tSD9000_Tot);
	GL_Variables.tSD9000_Totalizer_Value		:= Totalizer^;
	
	GL_Variables.SD9000_Flow_Value				:= GL_Variables.SD9000_Flow*0.1;
	GL_Variables.SD9000_Temp_Value				:= GL_Variables.SD9000_Temp/4*0.1;	// Right shift of 2
END_METHOD

END_FUNCTION_BLOCK

// Device/Application/Connected_Devices_Dashboard
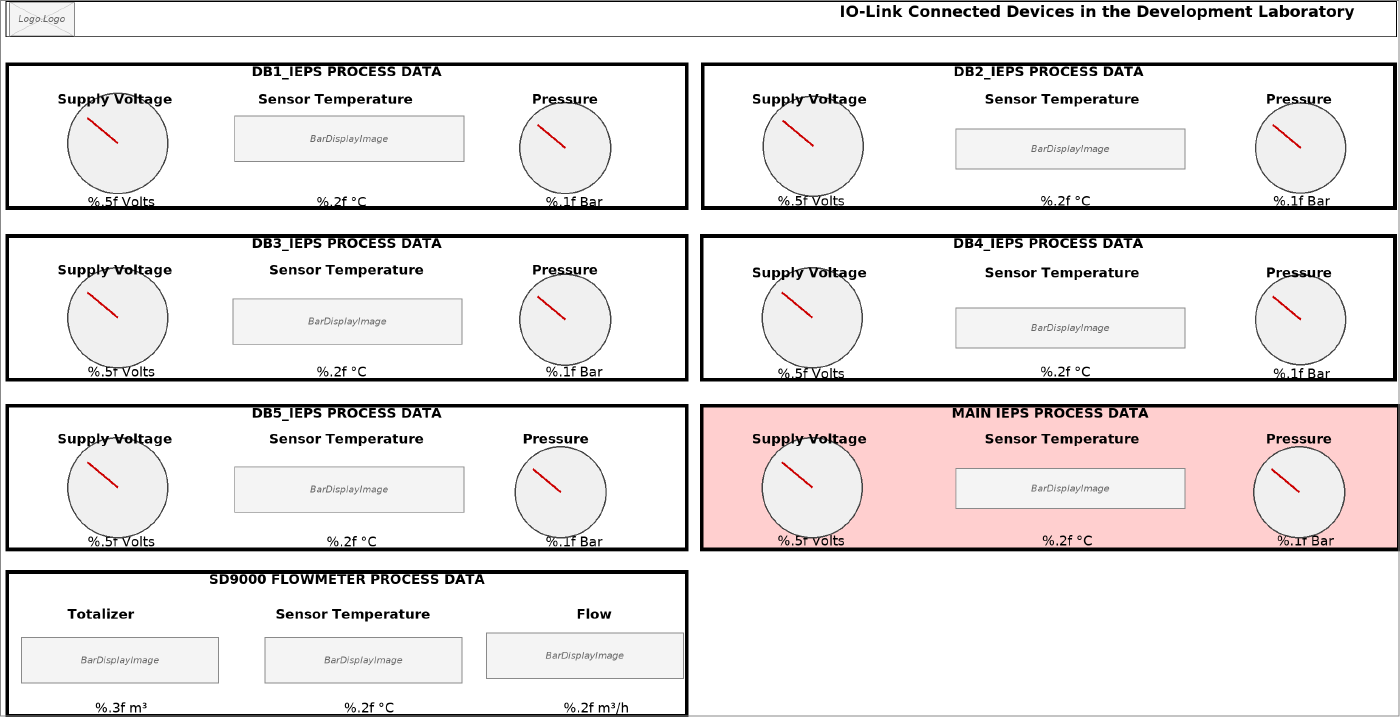
VISUALIZATION Connected_Devices_Dashboard  // 1524x781
    Rectangle (6,1 1514x39), "IO-Link Connected Devices in the Development Laboratory"
    Image (10,2 71x37), image: Logo.Logo
    Group (6,68 743x162)
        Rectangle (0,0 743x160), "DB1_IEPS PROCESS DATA"
        Meter360 (559,43 100x100), value: GL_Variables.pDB1_Pressure_Value, style: Meter-Meter360-Gray, scale format: %.0f, scale 0..10
            p518627256: bar
        Textfield (66,142 120x20), "%.5f Volts", text variable: GL_Variables.vDB1_Voltage_Value
        BarDisplayImage (249,58 250x50), value: GL_Variables.tDB1_Temp_Value, style: BarDisplayImage-Gray, scale format: %.0f, scale 20..50
        Textfield (306,142 120x20), "%.2f °C", text variable: GL_Variables.tDB1_Temp_Value
        Textfield (559,142 120x20), "%.1f Bar", text variable: GL_Variables.pDB1_Pressure_Value
        Meter180 (17,33 210x110), value: GL_Variables.vDB1_Voltage_Value, style: Meter-Meter180-Red, scale format: %.0f, scale 0..35
            p518627256: Volts
        Label (61,25 116x30), "Supply Voltage"
        Label (282,25 155x30), "Sensor Temperature"
        Label (559,25 100x30), "Pressure"
    Rectangle (6,255 743x160), "DB3_IEPS PROCESS DATA"
    Textfield (72,395 120x20), "%.5f Volts", text variable: GL_Variables.vDB3_Voltage_Value
    BarDisplayImage (253,325 250x50), value: GL_Variables.tDB3_Temp_Value, style: BarDisplayImage-Gray, scale format: %.0f, scale 20..50
    Textfield (312,395 120x20), "%.2f °C", text variable: GL_Variables.tDB3_Temp_Value
    Textfield (565,395 120x20), "%.1f Bar", text variable: GL_Variables.pDB3_Pressure_Value
    Meter180 (23,291 210x110), value: GL_Variables.vDB3_Voltage_Value, style: Meter-Meter180-Red, scale format: %.0f, scale 0..35
        p518627256: Volts
    Meter360 (565,298 100x100), value: GL_Variables.pDB3_Pressure_Value, style: Meter-Meter360-Gray, scale format: %.0f, scale 0..10
        p518627256: bar
    Label (67,279 116x30), "Supply Voltage"
    Label (300,279 155x30), "Sensor Temperature"
    Label (565,279 100x30), "Pressure"
    Group (6,440 743x160)
        Rectangle (0,0 743x160), "DB5_IEPS PROCESS DATA"
        Textfield (66,140 120x20), "%.5f Volts", text variable: GL_Variables.vDB5_Voltage_Value
        BarDisplayImage (249,68 250x50), value: GL_Variables.tDB5_Temp_Value, style: BarDisplayImage-Gray, scale format: %.0f, scale 20..50
        Textfield (317,140 120x20), "%.2f °C", text variable: GL_Variables.tDB5_Temp_Value
        Textfield (559,140 120x20), "%.1f Bar", text variable: GL_Variables.pDB5_Pressure_Value
        Meter180 (17,36 210x110), value: GL_Variables.vDB5_Voltage_Value, style: Meter-Meter180-Red, scale format: %.0f, scale 0..35
            p518627256: Volts
        Meter360 (549,46 110x100), value: GL_Variables.pDB5_Pressure_Value, style: Meter-Meter360-Gray, scale format: %.0f, scale 0..10
            p518627256: bar
        Label (61,23 116x30), "Supply Voltage"
        Label (294,23 155x30), "Sensor Temperature"
        Label (549,23 100x30), "Pressure"
    Group (763,68 757x161)
        Rectangle (0,0 757x160), "DB2_IEPS PROCESS DATA"
        Textfield (60,141 120x20), "%.5f Volts", text variable: GL_Variables.vDB2_Voltage_Value
        BarDisplayImage (277,72 250x44), value: GL_Variables.tDB2_Temp_Value, style: BarDisplayImage-Gray, scale format: %.0f, scale 20..50
        Textfield (337,141 120x20), "%.2f °C", text variable: GL_Variables.tDB2_Temp_Value
        Textfield (594,141 120x20), "%.1f Bar", text variable: GL_Variables.pDB2_Pressure_Value
        Meter180 (17,36 210x110), value: GL_Variables.vDB2_Voltage_Value, style: Meter-Meter180-Red, scale format: %.0f, scale 0..35
            p518627256: Volts
        Meter360 (603,43 99x100), value: GL_Variables.pDB2_Pressure_Value, style: Meter-Meter360-Gray, scale format: %.0f, scale 0..10
            p518627256: bar
        Label (60,25 116x30), "Supply Voltage"
        Label (316,25 155x30), "Sensor Temperature"
        Label (601,25 100x30), "Pressure"
    Group (762,255 758x162)
        Rectangle (0,0 758x160), "DB4_IEPS PROCESS DATA"
        Textfield (61,142 120x20), "%.5f Volts", text variable: GL_Variables.vDB4_Voltage_Value
        BarDisplayImage (278,80 250x44), value: GL_Variables.tDB4_Temp_Value, style: BarDisplayImage-Gray, scale format: %.0f, scale 20..50
        Textfield (338,140 120x20), "%.2f °C", text variable: GL_Variables.tDB4_Temp_Value
        Textfield (595,142 120x20), "%.1f Bar", text variable: GL_Variables.pDB4_Pressure_Value
        Meter180 (17,36 210x110), value: GL_Variables.vDB4_Voltage_Value, style: Meter-Meter180-Red, scale format: %.0f, scale 0..35
            p518627256: Volts
        Meter360 (604,43 99x100), value: GL_Variables.pDB4_Pressure_Value, style: Meter-Meter360-Gray, scale format: %.0f, scale 0..10
            p518627256: bar
        Label (61,27 116x30), "Supply Voltage"
        Label (317,27 155x30), "Sensor Temperature"
        Label (602,27 100x30), "Pressure"
    Group (762,440 762x160)
        Rectangle (0,0 762x160), "MAIN IEPS PROCESS DATA"
        Textfield (61,139 120x20), "%.5f Volts", text variable: GL_Variables.vDG_Voltage_Value
        BarDisplayImage (278,70 250x44), value: GL_Variables.tDG_Temp_Value, style: BarDisplayImage-Gray, scale format: %.0f, scale 20..50
        Textfield (340,139 120x20), "%.2f °C", text variable: GL_Variables.tDG_Temp_Value
        Textfield (599,139 120x20), "%.1f Bar", text variable: GL_Variables.pDG_Pressure_Value
        Meter180 (17,36 210x110), value: GL_Variables.vDG_Voltage_Value, style: Meter-Meter180-Red, scale format: %.0f, scale 0..35
            p518627256: Volts
        Meter360 (602,46 100x100), value: GL_Variables.pDG_Pressure_Value, style: Meter-Meter360-Gray, scale format: %.0f, scale 0..10
            p518627256: bar
        Label (61,23 116x30), "Supply Voltage"
        Label (317,23 155x30), "Sensor Temperature"
        Label (602,23 100x30), "Pressure"
    Group (6,621 743x160)
        Rectangle (0,0 743x160), "SD9000 FLOWMETER PROCESS DATA"
        Textfield (66,140 120x20), "%.3f m³", text variable: GL_Variables.tSD9000_Totalizer_Value
        BarDisplayImage (282,73 215x50), value: GL_Variables.SD9000_Temp_Value, style: BarDisplayImage-Gray, scale format: %.0f, scale 0..50
        Textfield (336,140 120x20), "%.2f °C", text variable: GL_Variables.SD9000_Temp_Value
        Textfield (583,140 120x20), "%.2f m³/h", text variable: GL_Variables.SD9000_Flow_value
        BarDisplayImage (523,68 215x50), value: GL_Variables.SD9000_Flow_value, style: BarDisplayImage-Gray, scale format: %.0f, scale 0..100
        BarDisplayImage (17,73 215x50), value: GL_Variables.tSD9000_Totalizer_Value, style: BarDisplayImage-Gray, scale format: %.0f, scale 0..1000
        Label (46,33 116x30), "Totalizer"
        Label (301,33 155x30), "Sensor Temperature"
        Label (583,33 116x30), "Flow"
END_VISUALIZATION
